FUNCTION_BLOCK "UTF8_TO_UNI"
{ S7_Optimized_Access := 'TRUE' }
VERSION : 0.1
   VAR_INPUT
      UTF8 : String[4];
   END_VAR

   VAR_OUTPUT
      UNICODE : Word;
   END_VAR

   VAR_TEMP
      TempDW : DWord;
      TempW : Array[0..3] of Word;
   END_VAR


BEGIN
	#TempDW := #UTF8[1];
	IF #TempDW < 16#80 THEN
	    #UNICODE := DWORD_TO_WORD(#TempDW AND 16#7F);
	ELSIF #TempDW >= 16#80 AND #TempDW < 16#C0 THEN
	    ;
	ELSIF #TempDW >= 16#C0 AND #TempDW < 16#E0 THEN
	    #TempDW := SHL(IN := #TempDW, N := 8);
	    #TempDW := #TempDW + BYTE_TO_WORD(#UTF8[2]);
	    #TempW[0] := DWORD_TO_WORD(SHR(IN:=#TempDW AND 16#1F00, N:=2));
	    #TempW[1] := DWORD_TO_WORD(#TempDW AND 16#3F);
	    #UNICODE := #TempW[0] + #TempW[1];
	ELSIF #TempDW >= 16#E0 AND #TempDW < 16#F0 THEN
	    #TempDW := SHL(IN := #TempDW, N := 8);
	    #TempDW := #TempDW + BYTE_TO_WORD(#UTF8[2]);
	    #TempDW := SHL(IN := #TempDW, N := 8);
	    #TempDW := #TempDW + BYTE_TO_WORD(#UTF8[3]);
	    #TempW[0] := DWORD_TO_WORD(SHR(IN:=#TempDW AND 16#0F0000, N:=4));
	    #TempW[1] := DWORD_TO_WORD(SHR(IN:=#TempDW AND 16#3F00, N:=2));
	    #TempW[2] := DWORD_TO_WORD(#TempDW AND 16#3F);
	    #UNICODE := #TempW[0] + #TempW[1] + #TempW[2];
	ELSIF #TempDW >= 16#F0 AND #TempDW < 16#F8 THEN
	    #TempDW := SHL(IN := #TempDW,  N := 8);
	    #TempDW := #TempDW + BYTE_TO_WORD(#UTF8[2]);
	    #TempDW := SHL(IN := #TempDW, N := 8);
	    #TempDW := #TempDW + BYTE_TO_WORD(#UTF8[3]);
	    #TempDW := SHL(IN := #TempDW,  N := 8);
	    #TempDW := #TempDW + BYTE_TO_WORD(#UTF8[4]);
	    #TempW[0] := DWORD_TO_WORD(SHR(IN:=#TempDW AND 16#7000000, N:=6));
	    #TempW[1] := DWORD_TO_WORD(SHR(IN:=#TempDW AND 16#3F0000, N:=4));
	    #TempW[2] := DWORD_TO_WORD(SHR(IN:=#TempDW AND 16#3F00, N:=2));
	    #TempW[3] := DWORD_TO_WORD(#TempDW AND 16#3F);
	    #UNICODE := #TempW[0] + #TempW[1] + #TempW[2] + #TempW[3];
	END_IF;
END_FUNCTION_BLOCK

FUNCTION_BLOCK "UNI_TO_GB2"
{ S7_Optimized_Access := 'TRUE' }
VERSION : 0.1
   VAR_INPUT
      UNICODE : Word;
   END_VAR

   VAR_OUTPUT
      GB2312 : Word;
   END_VAR

   VAR
      UNI : Array[0..7480] of Word := [16#00A4, 16#00A7, 16#00A8, 16#00B0, 16#00B1, 16#00B7, 16#00D7, 16#00E0, 16#00E1, 16#00E8, 16#00E9, 16#00EA, 16#00EC, 16#00ED, 16#00F2, 16#00F3, 16#00F7, 16#00F9, 16#00FA, 16#00FC, 16#0101, 16#0113, 16#011B, 16#012B, 16#0144, 16#0148, 16#014D, 16#016B, 16#01CE, 16#01D0, 16#01D2, 16#01D4, 16#01D6, 16#01D8, 16#01DA, 16#01DC, 16#0251, 16#0261, 16#02C7, 16#02C9, 16#0391, 16#0392, 16#0393, 16#0394, 16#0395, 16#0396, 16#0397, 16#0398, 16#0399, 16#039A, 16#039B, 16#039C, 16#039D, 16#039E, 16#039F, 16#03A0, 16#03A1, 16#03A3, 16#03A4, 16#03A5, 16#03A6, 16#03A7, 16#03A8, 16#03A9, 16#03B1, 16#03B2, 16#03B3, 16#03B4, 16#03B5, 16#03B6, 16#03B7, 16#03B8, 16#03B9, 16#03BA, 16#03BB, 16#03BC, 16#03BD, 16#03BE, 16#03BF, 16#03C0, 16#03C1, 16#03C3, 16#03C4, 16#03C5, 16#03C6, 16#03C7, 16#03C8, 16#03C9, 16#0401, 16#0410, 16#0411, 16#0412, 16#0413, 16#0414, 16#0415, 16#0416, 16#0417, 16#0418, 16#0419, 16#041A, 16#041B, 16#041C, 16#041D, 16#041E, 16#041F, 16#0420, 16#0421, 16#0422, 16#0423, 16#0424, 16#0425, 16#0426, 16#0427, 16#0428, 16#0429, 16#042A, 16#042B, 16#042C, 16#042D, 16#042E, 16#042F, 16#0430, 16#0431, 16#0432, 16#0433, 16#0434, 16#0435, 16#0436, 16#0437, 16#0438, 16#0439, 16#043A, 16#043B, 16#043C, 16#043D, 16#043E, 16#043F, 16#0440, 16#0441, 16#0442, 16#0443, 16#0444, 16#0445, 16#0446, 16#0447, 16#0448, 16#0449, 16#044A, 16#044B, 16#044C, 16#044D, 16#044E, 16#044F, 16#0451, 16#2014, 16#2016, 16#2018, 16#2019, 16#201C, 16#201D, 16#2026, 16#2030, 16#2032, 16#2033, 16#203B, 16#2103, 16#2116, 16#2160, 16#2161, 16#2162, 16#2163, 16#2164, 16#2165, 16#2166, 16#2167, 16#2168, 16#2169, 16#216A, 16#216B, 16#2170, 16#2171, 16#2172, 16#2173, 16#2174, 16#2175, 16#2176, 16#2177, 16#2178, 16#2179, 16#2190, 16#2191, 16#2192, 16#2193, 16#2208, 16#220F, 16#2211, 16#221A, 16#221D, 16#221E, 16#2220, 16#2225, 16#2227, 16#2228, 16#2229, 16#222A, 16#222B, 16#222E, 16#2234, 16#2235, 16#2236, 16#2237, 16#223D, 16#2248, 16#224C, 16#2260, 16#2261, 16#2264, 16#2265, 16#226E, 16#226F, 16#2299, 16#22A5, 16#2312, 16#2460, 16#2461, 16#2462, 16#2463, 16#2464, 16#2465, 16#2466, 16#2467, 16#2468, 16#2469, 16#2474, 16#2475, 16#2476, 16#2477, 16#2478, 16#2479, 16#247A, 16#247B, 16#247C, 16#247D, 16#247E, 16#247F, 16#2480, 16#2481, 16#2482, 16#2483, 16#2484, 16#2485, 16#2486, 16#2487, 16#2488, 16#2489, 16#248A, 16#248B, 16#248C, 16#248D, 16#248E, 16#248F, 16#2490, 16#2491, 16#2492, 16#2493, 16#2494, 16#2495, 16#2496, 16#2497, 16#2498, 16#2499, 16#249A, 16#249B, 16#2500, 16#2501, 16#2502, 16#2503, 16#2504, 16#2505, 16#2506, 16#2507, 16#2508, 16#2509, 16#250A, 16#250B, 16#250C, 16#250D, 16#250E, 16#250F, 16#2510, 16#2511, 16#2512, 16#2513, 16#2514, 16#2515, 16#2516, 16#2517, 16#2518, 16#2519, 16#251A, 16#251B, 16#251C, 16#251D, 16#251E, 16#251F, 16#2520, 16#2521, 16#2522, 16#2523, 16#2524, 16#2525, 16#2526, 16#2527, 16#2528, 16#2529, 16#252A, 16#252B, 16#252C, 16#252D, 16#252E, 16#252F, 16#2530, 16#2531, 16#2532, 16#2533, 16#2534, 16#2535, 16#2536, 16#2537, 16#2538, 16#2539, 16#253A, 16#253B, 16#253C, 16#253D, 16#253E, 16#253F, 16#2540, 16#2541, 16#2542, 16#2543, 16#2544, 16#2545, 16#2546, 16#2547, 16#2548, 16#2549, 16#254A, 16#254B, 16#25A0, 16#25A1, 16#25B2, 16#25B3, 16#25C6, 16#25C7, 16#25CB, 16#25CE, 16#25CF, 16#2605, 16#2606, 16#2640, 16#2642, 16#3000, 16#3001, 16#3002, 16#3003, 16#3005, 16#3008, 16#3009, 16#300A, 16#300B, 16#300C, 16#300D, 16#300E, 16#300F, 16#3010, 16#3011, 16#3013, 16#3014, 16#3015, 16#3016, 16#3017, 16#3041, 16#3042, 16#3043, 16#3044, 16#3045, 16#3046, 16#3047, 16#3048, 16#3049, 16#304A, 16#304B, 16#304C, 16#304D, 16#304E, 16#304F, 16#3050, 16#3051, 16#3052, 16#3053, 16#3054, 16#3055, 16#3056, 16#3057, 16#3058, 16#3059, 16#305A, 16#305B, 16#305C, 16#305D, 16#305E, 16#305F, 16#3060, 16#3061, 16#3062, 16#3063, 16#3064, 16#3065, 16#3066, 16#3067, 16#3068, 16#3069, 16#306A, 16#306B, 16#306C, 16#306D, 16#306E, 16#306F, 16#3070, 16#3071, 16#3072, 16#3073, 16#3074, 16#3075, 16#3076, 16#3077, 16#3078, 16#3079, 16#307A, 16#307B, 16#307C, 16#307D, 16#307E, 16#307F, 16#3080, 16#3081, 16#3082, 16#3083, 16#3084, 16#3085, 16#3086, 16#3087, 16#3088, 16#3089, 16#308A, 16#308B, 16#308C, 16#308D, 16#308E, 16#308F, 16#3090, 16#3091, 16#3092, 16#3093, 16#30A1, 16#30A2, 16#30A3, 16#30A4, 16#30A5, 16#30A6, 16#30A7, 16#30A8, 16#30A9, 16#30AA, 16#30AB, 16#30AC, 16#30AD, 16#30AE, 16#30AF, 16#30B0, 16#30B1, 16#30B2, 16#30B3, 16#30B4, 16#30B5, 16#30B6, 16#30B7, 16#30B8, 16#30B9, 16#30BA, 16#30BB, 16#30BC, 16#30BD, 16#30BE, 16#30BF, 16#30C0, 16#30C1, 16#30C2, 16#30C3, 16#30C4, 16#30C5, 16#30C6, 16#30C7, 16#30C8, 16#30C9, 16#30CA, 16#30CB, 16#30CC, 16#30CD, 16#30CE, 16#30CF, 16#30D0, 16#30D1, 16#30D2, 16#30D3, 16#30D4, 16#30D5, 16#30D6, 16#30D7, 16#30D8, 16#30D9, 16#30DA, 16#30DB, 16#30DC, 16#30DD, 16#30DE, 16#30DF, 16#30E0, 16#30E1, 16#30E2, 16#30E3, 16#30E4, 16#30E5, 16#30E6, 16#30E7, 16#30E8, 16#30E9, 16#30EA, 16#30EB, 16#30EC, 16#30ED, 16#30EE, 16#30EF, 16#30F0, 16#30F1, 16#30F2, 16#30F3, 16#30F4, 16#30F5, 16#30F6, 16#3105, 16#3106, 16#3107, 16#3108, 16#3109, 16#310A, 16#310B, 16#310C, 16#310D, 16#310E, 16#310F, 16#3110, 16#3111, 16#3112, 16#3113, 16#3114, 16#3115, 16#3116, 16#3117, 16#3118, 16#3119, 16#311A, 16#311B, 16#311C, 16#311D, 16#311E, 16#311F, 16#3120, 16#3121, 16#3122, 16#3123, 16#3124, 16#3125, 16#3126, 16#3127, 16#3128, 16#3129, 16#3220, 16#3221, 16#3222, 16#3223, 16#3224, 16#3225, 16#3226, 16#3227, 16#3228, 16#3229, 16#4E00, 16#4E01, 16#4E03, 16#4E07, 16#4E08, 16#4E09, 16#4E0A, 16#4E0B, 16#4E0C, 16#4E0D, 16#4E0E, 16#4E10, 16#4E11, 16#4E13, 16#4E14, 16#4E15, 16#4E16, 16#4E18, 16#4E19, 16#4E1A, 16#4E1B, 16#4E1C, 16#4E1D, 16#4E1E, 16#4E22, 16#4E24, 16#4E25, 16#4E27, 16#4E28, 16#4E2A, 16#4E2B, 16#4E2C, 16#4E2D, 16#4E30, 16#4E32, 16#4E34, 16#4E36, 16#4E38, 16#4E39, 16#4E3A, 16#4E3B, 16#4E3D, 16#4E3E, 16#4E3F, 16#4E43, 16#4E45, 16#4E47, 16#4E48, 16#4E49, 16#4E4B, 16#4E4C, 16#4E4D, 16#4E4E, 16#4E4F, 16#4E50, 16#4E52, 16#4E53, 16#4E54, 16#4E56, 16#4E58, 16#4E59, 16#4E5C, 16#4E5D, 16#4E5E, 16#4E5F, 16#4E60, 16#4E61, 16#4E66, 16#4E69, 16#4E70, 16#4E71, 16#4E73, 16#4E7E, 16#4E86, 16#4E88, 16#4E89, 16#4E8B, 16#4E8C, 16#4E8D, 16#4E8E, 16#4E8F, 16#4E91, 16#4E92, 16#4E93, 16#4E94, 16#4E95, 16#4E98, 16#4E9A, 16#4E9B, 16#4E9F, 16#4EA0, 16#4EA1, 16#4EA2, 16#4EA4, 16#4EA5, 16#4EA6, 16#4EA7, 16#4EA8, 16#4EA9, 16#4EAB, 16#4EAC, 16#4EAD, 16#4EAE, 16#4EB2, 16#4EB3, 16#4EB5, 16#4EBA, 16#4EBB, 16#4EBF, 16#4EC0, 16#4EC1, 16#4EC2, 16#4EC3, 16#4EC4, 16#4EC5, 16#4EC6, 16#4EC7, 16#4EC9, 16#4ECA, 16#4ECB, 16#4ECD, 16#4ECE, 16#4ED1, 16#4ED3, 16#4ED4, 16#4ED5, 16#4ED6, 16#4ED7, 16#4ED8, 16#4ED9, 16#4EDD, 16#4EDE, 16#4EDF, 16#4EE1, 16#4EE3, 16#4EE4, 16#4EE5, 16#4EE8, 16#4EEA, 16#4EEB, 16#4EEC, 16#4EF0, 16#4EF2, 16#4EF3, 16#4EF5, 16#4EF6, 16#4EF7, 16#4EFB, 16#4EFD, 16#4EFF, 16#4F01, 16#4F09, 16#4F0A, 16#4F0D, 16#4F0E, 16#4F0F, 16#4F10, 16#4F11, 16#4F17, 16#4F18, 16#4F19, 16#4F1A, 16#4F1B, 16#4F1E, 16#4F1F, 16#4F20, 16#4F22, 16#4F24, 16#4F25, 16#4F26, 16#4F27, 16#4F2A, 16#4F2B, 16#4F2F, 16#4F30, 16#4F32, 16#4F34, 16#4F36, 16#4F38, 16#4F3A, 16#4F3C, 16#4F3D, 16#4F43, 16#4F46, 16#4F4D, 16#4F4E, 16#4F4F, 16#4F50, 16#4F51, 16#4F53, 16#4F55, 16#4F57, 16#4F58, 16#4F59, 16#4F5A, 16#4F5B, 16#4F5C, 16#4F5D, 16#4F5E, 16#4F5F, 16#4F60, 16#4F63, 16#4F64, 16#4F65, 16#4F67, 16#4F69, 16#4F6C, 16#4F6F, 16#4F70, 16#4F73, 16#4F74, 16#4F76, 16#4F7B, 16#4F7C, 16#4F7E, 16#4F7F, 16#4F83, 16#4F84, 16#4F88, 16#4F89, 16#4F8B, 16#4F8D, 16#4F8F, 16#4F91, 16#4F94, 16#4F97, 16#4F9B, 16#4F9D, 16#4FA0, 16#4FA3, 16#4FA5, 16#4FA6, 16#4FA7, 16#4FA8, 16#4FA9, 16#4FAA, 16#4FAC, 16#4FAE, 16#4FAF, 16#4FB5, 16#4FBF, 16#4FC3, 16#4FC4, 16#4FC5, 16#4FCA, 16#4FCE, 16#4FCF, 16#4FD0, 16#4FD1, 16#4FD7, 16#4FD8, 16#4FDA, 16#4FDC, 16#4FDD, 16#4FDE, 16#4FDF, 16#4FE1, 16#4FE3, 16#4FE6, 16#4FE8, 16#4FE9, 16#4FEA, 16#4FED, 16#4FEE, 16#4FEF, 16#4FF1, 16#4FF3, 16#4FF8, 16#4FFA, 16#4FFE, 16#500C, 16#500D, 16#500F, 16#5012, 16#5014, 16#5018, 16#5019, 16#501A, 16#501C, 16#501F, 16#5021, 16#5025, 16#5026, 16#5028, 16#5029, 16#502A, 16#502C, 16#502D, 16#502E, 16#503A, 16#503C, 16#503E, 16#5043, 16#5047, 16#5048, 16#504C, 16#504E, 16#504F, 16#5055, 16#505A, 16#505C, 16#5065, 16#506C, 16#5076, 16#5077, 16#507B, 16#507E, 16#507F, 16#5080, 16#5085, 16#5088, 16#508D, 16#50A3, 16#50A5, 16#50A7, 16#50A8, 16#50A9, 16#50AC, 16#50B2, 16#50BA, 16#50BB, 16#50CF, 16#50D6, 16#50DA, 16#50E6, 16#50E7, 16#50EC, 16#50ED, 16#50EE, 16#50F3, 16#50F5, 16#50FB, 16#5106, 16#5107, 16#510B, 16#5112, 16#5121, 16#513F, 16#5140, 16#5141, 16#5143, 16#5144, 16#5145, 16#5146, 16#5148, 16#5149, 16#514B, 16#514D, 16#5151, 16#5154, 16#5155, 16#5156, 16#515A, 16#515C, 16#5162, 16#5165, 16#5168, 16#516B, 16#516C, 16#516D, 16#516E, 16#5170, 16#5171, 16#5173, 16#5174, 16#5175, 16#5176, 16#5177, 16#5178, 16#5179, 16#517B, 16#517C, 16#517D, 16#5180, 16#5181, 16#5182, 16#5185, 16#5188, 16#5189, 16#518C, 16#518D, 16#5192, 16#5195, 16#5196, 16#5197, 16#5199, 16#519B, 16#519C, 16#51A0, 16#51A2, 16#51A4, 16#51A5, 16#51AB, 16#51AC, 16#51AF, 16#51B0, 16#51B1, 16#51B2, 16#51B3, 16#51B5, 16#51B6, 16#51B7, 16#51BB, 16#51BC, 16#51BD, 16#51C0, 16#51C4, 16#51C6, 16#51C7, 16#51C9, 16#51CB, 16#51CC, 16#51CF, 16#51D1, 16#51DB, 16#51DD, 16#51E0, 16#51E1, 16#51E4, 16#51EB, 16#51ED, 16#51EF, 16#51F0, 16#51F3, 16#51F5, 16#51F6, 16#51F8, 16#51F9, 16#51FA, 16#51FB, 16#51FC, 16#51FD, 16#51FF, 16#5200, 16#5201, 16#5202, 16#5203, 16#5206, 16#5207, 16#5208, 16#520A, 16#520D, 16#520E, 16#5211, 16#5212, 16#5216, 16#5217, 16#5218, 16#5219, 16#521A, 16#521B, 16#521D, 16#5220, 16#5224, 16#5228, 16#5229, 16#522B, 16#522D, 16#522E, 16#5230, 16#5233, 16#5236, 16#5237, 16#5238, 16#5239, 16#523A, 16#523B, 16#523D, 16#523F, 16#5240, 16#5241, 16#5242, 16#5243, 16#524A, 16#524C, 16#524D, 16#5250, 16#5251, 16#5254, 16#5256, 16#525C, 16#525E, 16#5261, 16#5265, 16#5267, 16#5269, 16#526A, 16#526F, 16#5272, 16#527D, 16#527F, 16#5281, 16#5282, 16#5288, 16#5290, 16#5293, 16#529B, 16#529D, 16#529E, 16#529F, 16#52A0, 16#52A1, 16#52A2, 16#52A3, 16#52A8, 16#52A9, 16#52AA, 16#52AB, 16#52AC, 16#52AD, 16#52B1, 16#52B2, 16#52B3, 16#52BE, 16#52BF, 16#52C3, 16#52C7, 16#52C9, 16#52CB, 16#52D0, 16#52D2, 16#52D6, 16#52D8, 16#52DF, 16#52E4, 16#52F0, 16#52F9, 16#52FA, 16#52FE, 16#52FF, 16#5300, 16#5305, 16#5306, 16#5308, 16#530D, 16#530F, 16#5310, 16#5315, 16#5316, 16#5317, 16#5319, 16#531A, 16#531D, 16#5320, 16#5321, 16#5323, 16#5326, 16#532A, 16#532E, 16#5339, 16#533A, 16#533B, 16#533E, 16#533F, 16#5341, 16#5343, 16#5345, 16#5347, 16#5348, 16#5349, 16#534A, 16#534E, 16#534F, 16#5351, 16#5352, 16#5353, 16#5355, 16#5356, 16#5357, 16#535A, 16#535C, 16#535E, 16#535F, 16#5360, 16#5361, 16#5362, 16#5363, 16#5364, 16#5366, 16#5367, 16#5369, 16#536B, 16#536E, 16#536F, 16#5370, 16#5371, 16#5373, 16#5374, 16#5375, 16#5377, 16#5378, 16#537A, 16#537F, 16#5382, 16#5384, 16#5385, 16#5386, 16#5389, 16#538B, 16#538C, 16#538D, 16#5395, 16#5398, 16#539A, 16#539D, 16#539F, 16#53A2, 16#53A3, 16#53A5, 16#53A6, 16#53A8, 16#53A9, 16#53AE, 16#53B6, 16#53BB, 16#53BF, 16#53C1, 16#53C2, 16#53C8, 16#53C9, 16#53CA, 16#53CB, 16#53CC, 16#53CD, 16#53D1, 16#53D4, 16#53D6, 16#53D7, 16#53D8, 16#53D9, 16#53DB, 16#53DF, 16#53E0, 16#53E3, 16#53E4, 16#53E5, 16#53E6, 16#53E8, 16#53E9, 16#53EA, 16#53EB, 16#53EC, 16#53ED, 16#53EE, 16#53EF, 16#53F0, 16#53F1, 16#53F2, 16#53F3, 16#53F5, 16#53F6, 16#53F7, 16#53F8, 16#53F9, 16#53FB, 16#53FC, 16#53FD, 16#5401, 16#5403, 16#5404, 16#5406, 16#5408, 16#5409, 16#540A, 16#540C, 16#540D, 16#540E, 16#540F, 16#5410, 16#5411, 16#5412, 16#5413, 16#5415, 16#5416, 16#5417, 16#541B, 16#541D, 16#541E, 16#541F, 16#5420, 16#5421, 16#5423, 16#5426, 16#5427, 16#5428, 16#5429, 16#542B, 16#542C, 16#542D, 16#542E, 16#542F, 16#5431, 16#5432, 16#5434, 16#5435, 16#5438, 16#5439, 16#543B, 16#543C, 16#543E, 16#5440, 16#5443, 16#5446, 16#5448, 16#544A, 16#544B, 16#5450, 16#5452, 16#5453, 16#5454, 16#5455, 16#5456, 16#5457, 16#5458, 16#5459, 16#545B, 16#545C, 16#5462, 16#5464, 16#5466, 16#5468, 16#5471, 16#5472, 16#5473, 16#5475, 16#5476, 16#5477, 16#5478, 16#547B, 16#547C, 16#547D, 16#5480, 16#5482, 16#5484, 16#5486, 16#548B, 16#548C, 16#548E, 16#548F, 16#5490, 16#5492, 16#5494, 16#5495, 16#5496, 16#5499, 16#549A, 16#549B, 16#549D, 16#54A3, 16#54A4, 16#54A6, 16#54A7, 16#54A8, 16#54A9, 16#54AA, 16#54AB, 16#54AC, 16#54AD, 16#54AF, 16#54B1, 16#54B3, 16#54B4, 16#54B8, 16#54BB, 16#54BD, 16#54BF, 16#54C0, 16#54C1, 16#54C2, 16#54C4, 16#54C6, 16#54C7, 16#54C8, 16#54C9, 16#54CC, 16#54CD, 16#54CE, 16#54CF, 16#54D0, 16#54D1, 16#54D2, 16#54D3, 16#54D4, 16#54D5, 16#54D7, 16#54D9, 16#54DA, 16#54DC, 16#54DD, 16#54DE, 16#54DF, 16#54E5, 16#54E6, 16#54E7, 16#54E8, 16#54E9, 16#54EA, 16#54ED, 16#54EE, 16#54F2, 16#54F3, 16#54FA, 16#54FC, 16#54FD, 16#54FF, 16#5501, 16#5506, 16#5507, 16#5509, 16#550F, 16#5510, 16#5511, 16#5514, 16#551B, 16#5520, 16#5522, 16#5523, 16#5524, 16#5527, 16#552A, 16#552C, 16#552E, 16#552F, 16#5530, 16#5531, 16#5533, 16#5537, 16#553C, 16#553E, 16#553F, 16#5541, 16#5543, 16#5544, 16#5546, 16#5549, 16#554A, 16#5550, 16#5555, 16#5556, 16#555C, 16#5561, 16#5564, 16#5565, 16#5566, 16#5567, 16#556A, 16#556C, 16#556D, 16#556E, 16#5575, 16#5576, 16#5577, 16#5578, 16#557B, 16#557C, 16#557E, 16#5580, 16#5581, 16#5582, 16#5583, 16#5584, 16#5587, 16#5588, 16#5589, 16#558A, 16#558B, 16#558F, 16#5591, 16#5594, 16#5598, 16#5599, 16#559C, 16#559D, 16#559F, 16#55A7, 16#55B1, 16#55B3, 16#55B5, 16#55B7, 16#55B9, 16#55BB, 16#55BD, 16#55BE, 16#55C4, 16#55C5, 16#55C9, 16#55CC, 16#55CD, 16#55D1, 16#55D2, 16#55D3, 16#55D4, 16#55D6, 16#55DC, 16#55DD, 16#55DF, 16#55E1, 16#55E3, 16#55E4, 16#55E5, 16#55E6, 16#55E8, 16#55EA, 16#55EB, 16#55EC, 16#55EF, 16#55F2, 16#55F3, 16#55F5, 16#55F7, 16#55FD, 16#55FE, 16#5600, 16#5601, 16#5608, 16#5609, 16#560C, 16#560E, 16#560F, 16#5618, 16#561B, 16#561E, 16#561F, 16#5623, 16#5624, 16#5627, 16#562C, 16#562D, 16#5631, 16#5632, 16#5634, 16#5636, 16#5639, 16#563B, 16#563F, 16#564C, 16#564D, 16#564E, 16#5654, 16#5657, 16#5658, 16#5659, 16#565C, 16#5662, 16#5664, 16#5668, 16#5669, 16#566A, 16#566B, 16#566C, 16#5671, 16#5676, 16#567B, 16#567C, 16#5685, 16#5686, 16#568E, 16#568F, 16#5693, 16#56A3, 16#56AF, 16#56B7, 16#56BC, 16#56CA, 16#56D4, 16#56D7, 16#56DA, 16#56DB, 16#56DD, 16#56DE, 16#56DF, 16#56E0, 16#56E1, 16#56E2, 16#56E4, 16#56EB, 16#56ED, 16#56F0, 16#56F1, 16#56F4, 16#56F5, 16#56F9, 16#56FA, 16#56FD, 16#56FE, 16#56FF, 16#5703, 16#5704, 16#5706, 16#5708, 16#5709, 16#570A, 16#571C, 16#571F, 16#5723, 16#5728, 16#5729, 16#572A, 16#572C, 16#572D, 16#572E, 16#572F, 16#5730, 16#5733, 16#5739, 16#573A, 16#573B, 16#573E, 16#5740, 16#5742, 16#5747, 16#574A, 16#574C, 16#574D, 16#574E, 16#574F, 16#5750, 16#5751, 16#5757, 16#575A, 16#575B, 16#575C, 16#575D, 16#575E, 16#575F, 16#5760, 16#5761, 16#5764, 16#5766, 16#5768, 16#5769, 16#576A, 16#576B, 16#576D, 16#576F, 16#5773, 16#5776, 16#5777, 16#577B, 16#577C, 16#5782, 16#5783, 16#5784, 16#5785, 16#5786, 16#578B, 16#578C, 16#5792, 16#5793, 16#579B, 16#57A0, 16#57A1, 16#57A2, 16#57A3, 16#57A4, 16#57A6, 16#57A7, 16#57A9, 16#57AB, 16#57AD, 16#57AE, 16#57B2, 16#57B4, 16#57B8, 16#57C2, 16#57C3, 16#57CB, 16#57CE, 16#57CF, 16#57D2, 16#57D4, 16#57D5, 16#57D8, 16#57D9, 16#57DA, 16#57DD, 16#57DF, 16#57E0, 16#57E4, 16#57ED, 16#57EF, 16#57F4, 16#57F8, 16#57F9, 16#57FA, 16#57FD, 16#5800, 16#5802, 16#5806, 16#5807, 16#580B, 16#580D, 16#5811, 16#5815, 16#5819, 16#581E, 16#5820, 16#5821, 16#5824, 16#582A, 16#5830, 16#5835, 16#5844, 16#584C, 16#584D, 16#5851, 16#5854, 16#5858, 16#585E, 16#5865, 16#586B, 16#586C, 16#587E, 16#5880, 16#5881, 16#5883, 16#5885, 16#5889, 16#5892, 16#5893, 16#5899, 16#589A, 16#589E, 16#589F, 16#58A8, 16#58A9, 16#58BC, 16#58C1, 16#58C5, 16#58D1, 16#58D5, 16#58E4, 16#58EB, 16#58EC, 16#58EE, 16#58F0, 16#58F3, 16#58F6, 16#58F9, 16#5902, 16#5904, 16#5907, 16#590D, 16#590F, 16#5914, 16#5915, 16#5916, 16#5919, 16#591A, 16#591C, 16#591F, 16#5924, 16#5925, 16#5927, 16#5929, 16#592A, 16#592B, 16#592D, 16#592E, 16#592F, 16#5931, 16#5934, 16#5937, 16#5938, 16#5939, 16#593A, 16#593C, 16#5941, 16#5942, 16#5944, 16#5947, 16#5948, 16#5949, 16#594B, 16#594E, 16#594F, 16#5951, 16#5954, 16#5955, 16#5956, 16#5957, 16#5958, 16#595A, 16#5960, 16#5962, 16#5965, 16#5973, 16#5974, 16#5976, 16#5978, 16#5979, 16#597D, 16#5981, 16#5982, 16#5983, 16#5984, 16#5986, 16#5987, 16#5988, 16#598A, 16#598D, 16#5992, 16#5993, 16#5996, 16#5997, 16#5999, 16#599E, 16#59A3, 16#59A4, 16#59A5, 16#59A8, 16#59A9, 16#59AA, 16#59AB, 16#59AE, 16#59AF, 16#59B2, 16#59B9, 16#59BB, 16#59BE, 16#59C6, 16#59CA, 16#59CB, 16#59D0, 16#59D1, 16#59D2, 16#59D3, 16#59D4, 16#59D7, 16#59D8, 16#59DA, 16#59DC, 16#59DD, 16#59E3, 16#59E5, 16#59E8, 16#59EC, 16#59F9, 16#59FB, 16#59FF, 16#5A01, 16#5A03, 16#5A04, 16#5A05, 16#5A06, 16#5A07, 16#5A08, 16#5A09, 16#5A0C, 16#5A11, 16#5A13, 16#5A18, 16#5A1C, 16#5A1F, 16#5A20, 16#5A23, 16#5A25, 16#5A29, 16#5A31, 16#5A32, 16#5A34, 16#5A36, 16#5A3C, 16#5A40, 16#5A46, 16#5A49, 16#5A4A, 16#5A55, 16#5A5A, 16#5A62, 16#5A67, 16#5A6A, 16#5A74, 16#5A75, 16#5A76, 16#5A77, 16#5A7A, 16#5A7F, 16#5A92, 16#5A9A, 16#5A9B, 16#5AAA, 16#5AB2, 16#5AB3, 16#5AB5, 16#5AB8, 16#5ABE, 16#5AC1, 16#5AC2, 16#5AC9, 16#5ACC, 16#5AD2, 16#5AD4, 16#5AD6, 16#5AD8, 16#5ADC, 16#5AE0, 16#5AE1, 16#5AE3, 16#5AE6, 16#5AE9, 16#5AEB, 16#5AF1, 16#5B09, 16#5B16, 16#5B17, 16#5B32, 16#5B34, 16#5B37, 16#5B40, 16#5B50, 16#5B51, 16#5B53, 16#5B54, 16#5B55, 16#5B57, 16#5B58, 16#5B59, 16#5B5A, 16#5B5B, 16#5B5C, 16#5B5D, 16#5B5F, 16#5B62, 16#5B63, 16#5B64, 16#5B65, 16#5B66, 16#5B69, 16#5B6A, 16#5B6C, 16#5B70, 16#5B71, 16#5B73, 16#5B75, 16#5B7A, 16#5B7D, 16#5B80, 16#5B81, 16#5B83, 16#5B84, 16#5B85, 16#5B87, 16#5B88, 16#5B89, 16#5B8B, 16#5B8C, 16#5B8F, 16#5B93, 16#5B95, 16#5B97, 16#5B98, 16#5B99, 16#5B9A, 16#5B9B, 16#5B9C, 16#5B9D, 16#5B9E, 16#5BA0, 16#5BA1, 16#5BA2, 16#5BA3, 16#5BA4, 16#5BA5, 16#5BA6, 16#5BAA, 16#5BAB, 16#5BB0, 16#5BB3, 16#5BB4, 16#5BB5, 16#5BB6, 16#5BB8, 16#5BB9, 16#5BBD, 16#5BBE, 16#5BBF, 16#5BC2, 16#5BC4, 16#5BC5, 16#5BC6, 16#5BC7, 16#5BCC, 16#5BD0, 16#5BD2, 16#5BD3, 16#5BDD, 16#5BDE, 16#5BDF, 16#5BE1, 16#5BE4, 16#5BE5, 16#5BE8, 16#5BEE, 16#5BF0, 16#5BF8, 16#5BF9, 16#5BFA, 16#5BFB, 16#5BFC, 16#5BFF, 16#5C01, 16#5C04, 16#5C06, 16#5C09, 16#5C0A, 16#5C0F, 16#5C11, 16#5C14, 16#5C15, 16#5C16, 16#5C18, 16#5C1A, 16#5C1C, 16#5C1D, 16#5C22, 16#5C24, 16#5C25, 16#5C27, 16#5C2C, 16#5C31, 16#5C34, 16#5C38, 16#5C39, 16#5C3A, 16#5C3B, 16#5C3C, 16#5C3D, 16#5C3E, 16#5C3F, 16#5C40, 16#5C41, 16#5C42, 16#5C45, 16#5C48, 16#5C49, 16#5C4A, 16#5C4B, 16#5C4E, 16#5C4F, 16#5C50, 16#5C51, 16#5C55, 16#5C59, 16#5C5E, 16#5C60, 16#5C61, 16#5C63, 16#5C65, 16#5C66, 16#5C6E, 16#5C6F, 16#5C71, 16#5C79, 16#5C7A, 16#5C7F, 16#5C81, 16#5C82, 16#5C88, 16#5C8C, 16#5C8D, 16#5C90, 16#5C91, 16#5C94, 16#5C96, 16#5C97, 16#5C98, 16#5C99, 16#5C9A, 16#5C9B, 16#5C9C, 16#5CA2, 16#5CA3, 16#5CA9, 16#5CAB, 16#5CAC, 16#5CAD, 16#5CB1, 16#5CB3, 16#5CB5, 16#5CB7, 16#5CB8, 16#5CBD, 16#5CBF, 16#5CC1, 16#5CC4, 16#5CCB, 16#5CD2, 16#5CD9, 16#5CE1, 16#5CE4, 16#5CE5, 16#5CE6, 16#5CE8, 16#5CEA, 16#5CED, 16#5CF0, 16#5CFB, 16#5D02, 16#5D03, 16#5D06, 16#5D07, 16#5D0E, 16#5D14, 16#5D16, 16#5D1B, 16#5D1E, 16#5D24, 16#5D26, 16#5D27, 16#5D29, 16#5D2D, 16#5D2E, 16#5D34, 16#5D3D, 16#5D3E, 16#5D47, 16#5D4A, 16#5D4B, 16#5D4C, 16#5D58, 16#5D5B, 16#5D5D, 16#5D69, 16#5D6B, 16#5D6C, 16#5D6F, 16#5D74, 16#5D82, 16#5D99, 16#5D9D, 16#5DB7, 16#5DC5, 16#5DCD, 16#5DDB, 16#5DDD, 16#5DDE, 16#5DE1, 16#5DE2, 16#5DE5, 16#5DE6, 16#5DE7, 16#5DE8, 16#5DE9, 16#5DEB, 16#5DEE, 16#5DEF, 16#5DF1, 16#5DF2, 16#5DF3, 16#5DF4, 16#5DF7, 16#5DFD, 16#5DFE, 16#5E01, 16#5E02, 16#5E03, 16#5E05, 16#5E06, 16#5E08, 16#5E0C, 16#5E0F, 16#5E10, 16#5E11, 16#5E14, 16#5E15, 16#5E16, 16#5E18, 16#5E19, 16#5E1A, 16#5E1B, 16#5E1C, 16#5E1D, 16#5E26, 16#5E27, 16#5E2D, 16#5E2E, 16#5E31, 16#5E37, 16#5E38, 16#5E3B, 16#5E3C, 16#5E3D, 16#5E42, 16#5E44, 16#5E45, 16#5E4C, 16#5E54, 16#5E55, 16#5E5B, 16#5E5E, 16#5E61, 16#5E62, 16#5E72, 16#5E73, 16#5E74, 16#5E76, 16#5E78, 16#5E7A, 16#5E7B, 16#5E7C, 16#5E7D, 16#5E7F, 16#5E80, 16#5E84, 16#5E86, 16#5E87, 16#5E8A, 16#5E8B, 16#5E8F, 16#5E90, 16#5E91, 16#5E93, 16#5E94, 16#5E95, 16#5E96, 16#5E97, 16#5E99, 16#5E9A, 16#5E9C, 16#5E9E, 16#5E9F, 16#5EA0, 16#5EA5, 16#5EA6, 16#5EA7, 16#5EAD, 16#5EB3, 16#5EB5, 16#5EB6, 16#5EB7, 16#5EB8, 16#5EB9, 16#5EBE, 16#5EC9, 16#5ECA, 16#5ED1, 16#5ED2, 16#5ED3, 16#5ED6, 16#5EDB, 16#5EE8, 16#5EEA, 16#5EF4, 16#5EF6, 16#5EF7, 16#5EFA, 16#5EFE, 16#5EFF, 16#5F00, 16#5F01, 16#5F02, 16#5F03, 16#5F04, 16#5F08, 16#5F0A, 16#5F0B, 16#5F0F, 16#5F11, 16#5F13, 16#5F15, 16#5F17, 16#5F18, 16#5F1B, 16#5F1F, 16#5F20, 16#5F25, 16#5F26, 16#5F27, 16#5F29, 16#5F2A, 16#5F2D, 16#5F2F, 16#5F31, 16#5F39, 16#5F3A, 16#5F3C, 16#5F40, 16#5F50, 16#5F52, 16#5F53, 16#5F55, 16#5F56, 16#5F57, 16#5F58, 16#5F5D, 16#5F61, 16#5F62, 16#5F64, 16#5F66, 16#5F69, 16#5F6A, 16#5F6C, 16#5F6D, 16#5F70, 16#5F71, 16#5F73, 16#5F77, 16#5F79, 16#5F7B, 16#5F7C, 16#5F80, 16#5F81, 16#5F82, 16#5F84, 16#5F85, 16#5F87, 16#5F88, 16#5F89, 16#5F8A, 16#5F8B, 16#5F8C, 16#5F90, 16#5F92, 16#5F95, 16#5F97, 16#5F98, 16#5F99, 16#5F9C, 16#5FA1, 16#5FA8, 16#5FAA, 16#5FAD, 16#5FAE, 16#5FB5, 16#5FB7, 16#5FBC, 16#5FBD, 16#5FC3, 16#5FC4, 16#5FC5, 16#5FC6, 16#5FC9, 16#5FCC, 16#5FCD, 16#5FCF, 16#5FD0, 16#5FD1, 16#5FD2, 16#5FD6, 16#5FD7, 16#5FD8, 16#5FD9, 16#5FDD, 16#5FE0, 16#5FE1, 16#5FE4, 16#5FE7, 16#5FEA, 16#5FEB, 16#5FED, 16#5FEE, 16#5FF1, 16#5FF5, 16#5FF8, 16#5FFB, 16#5FFD, 16#5FFE, 16#5FFF, 16#6000, 16#6001, 16#6002, 16#6003, 16#6004, 16#6005, 16#6006, 16#600A, 16#600D, 16#600E, 16#600F, 16#6012, 16#6014, 16#6015, 16#6016, 16#6019, 16#601B, 16#601C, 16#601D, 16#6020, 16#6021, 16#6025, 16#6026, 16#6027, 16#6028, 16#6029, 16#602A, 16#602B, 16#602F, 16#6035, 16#603B, 16#603C, 16#603F, 16#6041, 16#6042, 16#6043, 16#604B, 16#604D, 16#6050, 16#6052, 16#6055, 16#6059, 16#605A, 16#605D, 16#6062, 16#6063, 16#6064, 16#6067, 16#6068, 16#6069, 16#606A, 16#606B, 16#606C, 16#606D, 16#606F, 16#6070, 16#6073, 16#6076, 16#6078, 16#6079, 16#607A, 16#607B, 16#607C, 16#607D, 16#607F, 16#6083, 16#6084, 16#6089, 16#608C, 16#608D, 16#6092, 16#6094, 16#6096, 16#609A, 16#609B, 16#609D, 16#609F, 16#60A0, 16#60A3, 16#60A6, 16#60A8, 16#60AB, 16#60AC, 16#60AD, 16#60AF, 16#60B1, 16#60B2, 16#60B4, 16#60B8, 16#60BB, 16#60BC, 16#60C5, 16#60C6, 16#60CA, 16#60CB, 16#60D1, 16#60D5, 16#60D8, 16#60DA, 16#60DC, 16#60DD, 16#60DF, 16#60E0, 16#60E6, 16#60E7, 16#60E8, 16#60E9, 16#60EB, 16#60EC, 16#60ED, 16#60EE, 16#60EF, 16#60F0, 16#60F3, 16#60F4, 16#60F6, 16#60F9, 16#60FA, 16#6100, 16#6101, 16#6106, 16#6108, 16#6109, 16#610D, 16#610E, 16#610F, 16#6115, 16#611A, 16#611F, 16#6120, 16#6123, 16#6124, 16#6126, 16#6127, 16#612B, 16#613F, 16#6148, 16#614A, 16#614C, 16#614E, 16#6151, 16#6155, 16#615D, 16#6162, 16#6167, 16#6168, 16#6170, 16#6175, 16#6177, 16#618B, 16#618E, 16#6194, 16#619D, 16#61A7, 16#61A8, 16#61A9, 16#61AC, 16#61B7, 16#61BE, 16#61C2, 16#61C8, 16#61CA, 16#61CB, 16#61D1, 16#61D2, 16#61D4, 16#61E6, 16#61F5, 16#61FF, 16#6206, 16#6208, 16#620A, 16#620B, 16#620C, 16#620D, 16#620E, 16#620F, 16#6210, 16#6211, 16#6212, 16#6215, 16#6216, 16#6217, 16#6218, 16#621A, 16#621B, 16#621F, 16#6221, 16#6222, 16#6224, 16#6225, 16#622A, 16#622C, 16#622E, 16#6233, 16#6234, 16#6237, 16#623D, 16#623E, 16#623F, 16#6240, 16#6241, 16#6243, 16#6247, 16#6248, 16#6249, 16#624B, 16#624C, 16#624D, 16#624E, 16#6251, 16#6252, 16#6253, 16#6254, 16#6258, 16#625B, 16#6263, 16#6266, 16#6267, 16#6269, 16#626A, 16#626B, 16#626C, 16#626D, 16#626E, 16#626F, 16#6270, 16#6273, 16#6276, 16#6279, 16#627C, 16#627E, 16#627F, 16#6280, 16#6284, 16#6289, 16#628A, 16#6291, 16#6292, 16#6293, 16#6295, 16#6296, 16#6297, 16#6298, 16#629A, 16#629B, 16#629F, 16#62A0, 16#62A1, 16#62A2, 16#62A4, 16#62A5, 16#62A8, 16#62AB, 16#62AC, 16#62B1, 16#62B5, 16#62B9, 16#62BB, 16#62BC, 16#62BD, 16#62BF, 16#62C2, 16#62C4, 16#62C5, 16#62C6, 16#62C7, 16#62C8, 16#62C9, 16#62CA, 16#62CC, 16#62CD, 16#62CE, 16#62D0, 16#62D2, 16#62D3, 16#62D4, 16#62D6, 16#62D7, 16#62D8, 16#62D9, 16#62DA, 16#62DB, 16#62DC, 16#62DF, 16#62E2, 16#62E3, 16#62E5, 16#62E6, 16#62E7, 16#62E8, 16#62E9, 16#62EC, 16#62ED, 16#62EE, 16#62EF, 16#62F1, 16#62F3, 16#62F4, 16#62F6, 16#62F7, 16#62FC, 16#62FD, 16#62FE, 16#62FF, 16#6301, 16#6302, 16#6307, 16#6308, 16#6309, 16#630E, 16#6311, 16#6316, 16#631A, 16#631B, 16#631D, 16#631E, 16#631F, 16#6320, 16#6321, 16#6322, 16#6323, 16#6324, 16#6325, 16#6328, 16#632A, 16#632B, 16#632F, 16#6332, 16#6339, 16#633A, 16#633D, 16#6342, 16#6343, 16#6345, 16#6346, 16#6349, 16#634B, 16#634C, 16#634D, 16#634E, 16#634F, 16#6350, 16#6355, 16#635E, 16#635F, 16#6361, 16#6362, 16#6363, 16#6367, 16#6369, 16#636D, 16#636E, 16#6371, 16#6376, 16#6377, 16#637A, 16#637B, 16#6380, 16#6382, 16#6387, 16#6388, 16#6389, 16#638A, 16#638C, 16#638E, 16#638F, 16#6390, 16#6392, 16#6396, 16#6398, 16#63A0, 16#63A2, 16#63A3, 16#63A5, 16#63A7, 16#63A8, 16#63A9, 16#63AA, 16#63AC, 16#63AD, 16#63AE, 16#63B0, 16#63B3, 16#63B4, 16#63B7, 16#63B8, 16#63BA, 16#63BC, 16#63BE, 16#63C4, 16#63C6, 16#63C9, 16#63CD, 16#63CE, 16#63CF, 16#63D0, 16#63D2, 16#63D6, 16#63DE, 16#63E0, 16#63E1, 16#63E3, 16#63E9, 16#63EA, 16#63ED, 16#63F2, 16#63F4, 16#63F6, 16#63F8, 16#63FD, 16#63FF, 16#6400, 16#6401, 16#6402, 16#6405, 16#640B, 16#640C, 16#640F, 16#6410, 16#6413, 16#6414, 16#641B, 16#641C, 16#641E, 16#6420, 16#6421, 16#6426, 16#642A, 16#642C, 16#642D, 16#6434, 16#643A, 16#643D, 16#643F, 16#6441, 16#6444, 16#6445, 16#6446, 16#6447, 16#6448, 16#644A, 16#6452, 16#6454, 16#6458, 16#645E, 16#6467, 16#6469, 16#646D, 16#6478, 16#6479, 16#647A, 16#6482, 16#6484, 16#6485, 16#6487, 16#6491, 16#6492, 16#6495, 16#6496, 16#6499, 16#649E, 16#64A4, 16#64A9, 16#64AC, 16#64AD, 16#64AE, 16#64B0, 16#64B5, 16#64B7, 16#64B8, 16#64BA, 16#64BC, 16#64C0, 16#64C2, 16#64C5, 16#64CD, 16#64CE, 16#64D0, 16#64D2, 16#64D7, 16#64D8, 16#64DE, 16#64E2, 16#64E4, 16#64E6, 16#6500, 16#6509, 16#6512, 16#6518, 16#6525, 16#652B, 16#652E, 16#652F, 16#6534, 16#6535, 16#6536, 16#6538, 16#6539, 16#653B, 16#653E, 16#653F, 16#6545, 16#6548, 16#6549, 16#654C, 16#654F, 16#6551, 16#6555, 16#6556, 16#6559, 16#655B, 16#655D, 16#655E, 16#6562, 16#6563, 16#6566, 16#656B, 16#656C, 16#6570, 16#6572, 16#6574, 16#6577, 16#6587, 16#658B, 16#658C, 16#6590, 16#6591, 16#6593, 16#6597, 16#6599, 16#659B, 16#659C, 16#659F, 16#65A1, 16#65A4, 16#65A5, 16#65A7, 16#65A9, 16#65AB, 16#65AD, 16#65AF, 16#65B0, 16#65B9, 16#65BC, 16#65BD, 16#65C1, 16#65C3, 16#65C4, 16#65C5, 16#65C6, 16#65CB, 16#65CC, 16#65CE, 16#65CF, 16#65D2, 16#65D6, 16#65D7, 16#65E0, 16#65E2, 16#65E5, 16#65E6, 16#65E7, 16#65E8, 16#65E9, 16#65EC, 16#65ED, 16#65EE, 16#65EF, 16#65F0, 16#65F1, 16#65F6, 16#65F7, 16#65FA, 16#6600, 16#6602, 16#6603, 16#6606, 16#660A, 16#660C, 16#660E, 16#660F, 16#6613, 16#6614, 16#6615, 16#6619, 16#661D, 16#661F, 16#6620, 16#6625, 16#6627, 16#6628, 16#662D, 16#662F, 16#6631, 16#6634, 16#6635, 16#6636, 16#663C, 16#663E, 16#6641, 16#6643, 16#664B, 16#664C, 16#664F, 16#6652, 16#6653, 16#6654, 16#6655, 16#6656, 16#6657, 16#665A, 16#665F, 16#6661, 16#6664, 16#6666, 16#6668, 16#666E, 16#666F, 16#6670, 16#6674, 16#6676, 16#6677, 16#667A, 16#667E, 16#6682, 16#6684, 16#6687, 16#668C, 16#6691, 16#6696, 16#6697, 16#669D, 16#66A7, 16#66A8, 16#66AE, 16#66B4, 16#66B9, 16#66BE, 16#66D9, 16#66DB, 16#66DC, 16#66DD, 16#66E6, 16#66E9, 16#66F0, 16#66F2, 16#66F3, 16#66F4, 16#66F7, 16#66F9, 16#66FC, 16#66FE, 16#66FF, 16#6700, 16#6708, 16#6709, 16#670A, 16#670B, 16#670D, 16#6710, 16#6714, 16#6715, 16#6717, 16#671B, 16#671D, 16#671F, 16#6726, 16#6728, 16#672A, 16#672B, 16#672C, 16#672D, 16#672F, 16#6731, 16#6734, 16#6735, 16#673A, 16#673D, 16#6740, 16#6742, 16#6743, 16#6746, 16#6748, 16#6749, 16#674C, 16#674E, 16#674F, 16#6750, 16#6751, 16#6753, 16#6756, 16#675C, 16#675E, 16#675F, 16#6760, 16#6761, 16#6765, 16#6768, 16#6769, 16#676A, 16#676D, 16#676F, 16#6770, 16#6772, 16#6773, 16#6775, 16#6777, 16#677C, 16#677E, 16#677F, 16#6781, 16#6784, 16#6787, 16#6789, 16#678B, 16#6790, 16#6795, 16#6797, 16#6798, 16#679A, 16#679C, 16#679D, 16#679E, 16#67A2, 16#67A3, 16#67A5, 16#67A7, 16#67A8, 16#67AA, 16#67AB, 16#67AD, 16#67AF, 16#67B0, 16#67B3, 16#67B5, 16#67B6, 16#67B7, 16#67B8, 16#67C1, 16#67C3, 16#67C4, 16#67CF, 16#67D0, 16#67D1, 16#67D2, 16#67D3, 16#67D4, 16#67D8, 16#67D9, 16#67DA, 16#67DC, 16#67DD, 16#67DE, 16#67E0, 16#67E2, 16#67E5, 16#67E9, 16#67EC, 16#67EF, 16#67F0, 16#67F1, 16#67F3, 16#67F4, 16#67FD, 16#67FF, 16#6800, 16#6805, 16#6807, 16#6808, 16#6809, 16#680A, 16#680B, 16#680C, 16#680E, 16#680F, 16#6811, 16#6813, 16#6816, 16#6817, 16#681D, 16#6821, 16#6829, 16#682A, 16#6832, 16#6833, 16#6837, 16#6838, 16#6839, 16#683C, 16#683D, 16#683E, 16#6840, 16#6841, 16#6842, 16#6843, 16#6844, 16#6845, 16#6846, 16#6848, 16#6849, 16#684A, 16#684C, 16#684E, 16#6850, 16#6851, 16#6853, 16#6854, 16#6855, 16#6860, 16#6861, 16#6862, 16#6863, 16#6864, 16#6865, 16#6866, 16#6867, 16#6868, 16#6869, 16#686B, 16#6874, 16#6876, 16#6877, 16#6881, 16#6883, 16#6885, 16#6886, 16#688F, 16#6893, 16#6897, 16#68A2, 16#68A6, 16#68A7, 16#68A8, 16#68AD, 16#68AF, 16#68B0, 16#68B3, 16#68B5, 16#68C0, 16#68C2, 16#68C9, 16#68CB, 16#68CD, 16#68D2, 16#68D5, 16#68D8, 16#68DA, 16#68E0, 16#68E3, 16#68EE, 16#68F0, 16#68F1, 16#68F5, 16#68F9, 16#68FA, 16#68FC, 16#6901, 16#6905, 16#690B, 16#690D, 16#690E, 16#6910, 16#6912, 16#691F, 16#6920, 16#6924, 16#692D, 16#6930, 16#6934, 16#6939, 16#693D, 16#693F, 16#6942, 16#6954, 16#6957, 16#695A, 16#695D, 16#695E, 16#6960, 16#6963, 16#6966, 16#696B, 16#696E, 16#6971, 16#6977, 16#6978, 16#6979, 16#697C, 16#6980, 16#6982, 16#6984, 16#6986, 16#6987, 16#6988, 16#6989, 16#698D, 16#6994, 16#6995, 16#6998, 16#699B, 16#699C, 16#69A7, 16#69A8, 16#69AB, 16#69AD, 16#69B1, 16#69B4, 16#69B7, 16#69BB, 16#69C1, 16#69CA, 16#69CC, 16#69CE, 16#69D0, 16#69D4, 16#69DB, 16#69DF, 16#69E0, 16#69ED, 16#69F2, 16#69FD, 16#69FF, 16#6A0A, 16#6A17, 16#6A18, 16#6A1F, 16#6A21, 16#6A28, 16#6A2A, 16#6A2F, 16#6A31, 16#6A35, 16#6A3D, 16#6A3E, 16#6A44, 16#6A47, 16#6A50, 16#6A58, 16#6A59, 16#6A5B, 16#6A61, 16#6A65, 16#6A71, 16#6A79, 16#6A7C, 16#6A80, 16#6A84, 16#6A8E, 16#6A90, 16#6A91, 16#6A97, 16#6AA0, 16#6AA9, 16#6AAB, 16#6AAC, 16#6B20, 16#6B21, 16#6B22, 16#6B23, 16#6B24, 16#6B27, 16#6B32, 16#6B37, 16#6B39, 16#6B3A, 16#6B3E, 16#6B43, 16#6B46, 16#6B47, 16#6B49, 16#6B4C, 16#6B59, 16#6B62, 16#6B63, 16#6B64, 16#6B65, 16#6B66, 16#6B67, 16#6B6A, 16#6B79, 16#6B7B, 16#6B7C, 16#6B81, 16#6B82, 16#6B83, 16#6B84, 16#6B86, 16#6B87, 16#6B89, 16#6B8A, 16#6B8B, 16#6B8D, 16#6B92, 16#6B93, 16#6B96, 16#6B9A, 16#6B9B, 16#6BA1, 16#6BAA, 16#6BB3, 16#6BB4, 16#6BB5, 16#6BB7, 16#6BBF, 16#6BC1, 16#6BC2, 16#6BC5, 16#6BCB, 16#6BCD, 16#6BCF, 16#6BD2, 16#6BD3, 16#6BD4, 16#6BD5, 16#6BD6, 16#6BD7, 16#6BD9, 16#6BDB, 16#6BE1, 16#6BEA, 16#6BEB, 16#6BEF, 16#6BF3, 16#6BF5, 16#6BF9, 16#6BFD, 16#6C05, 16#6C06, 16#6C07, 16#6C0D, 16#6C0F, 16#6C10, 16#6C11, 16#6C13, 16#6C14, 16#6C15, 16#6C16, 16#6C18, 16#6C19, 16#6C1A, 16#6C1B, 16#6C1F, 16#6C21, 16#6C22, 16#6C24, 16#6C26, 16#6C27, 16#6C28, 16#6C29, 16#6C2A, 16#6C2E, 16#6C2F, 16#6C30, 16#6C32, 16#6C34, 16#6C35, 16#6C38, 16#6C3D, 16#6C40, 16#6C41, 16#6C42, 16#6C46, 16#6C47, 16#6C49, 16#6C4A, 16#6C50, 16#6C54, 16#6C55, 16#6C57, 16#6C5B, 16#6C5C, 16#6C5D, 16#6C5E, 16#6C5F, 16#6C60, 16#6C61, 16#6C64, 16#6C68, 16#6C69, 16#6C6A, 16#6C70, 16#6C72, 16#6C74, 16#6C76, 16#6C79, 16#6C7D, 16#6C7E, 16#6C81, 16#6C82, 16#6C83, 16#6C85, 16#6C86, 16#6C88, 16#6C89, 16#6C8C, 16#6C8F, 16#6C90, 16#6C93, 16#6C94, 16#6C99, 16#6C9B, 16#6C9F, 16#6CA1, 16#6CA3, 16#6CA4, 16#6CA5, 16#6CA6, 16#6CA7, 16#6CA9, 16#6CAA, 16#6CAB, 16#6CAD, 16#6CAE, 16#6CB1, 16#6CB2, 16#6CB3, 16#6CB8, 16#6CB9, 16#6CBB, 16#6CBC, 16#6CBD, 16#6CBE, 16#6CBF, 16#6CC4, 16#6CC5, 16#6CC9, 16#6CCA, 16#6CCC, 16#6CD0, 16#6CD3, 16#6CD4, 16#6CD5, 16#6CD6, 16#6CD7, 16#6CDB, 16#6CDE, 16#6CE0, 16#6CE1, 16#6CE2, 16#6CE3, 16#6CE5, 16#6CE8, 16#6CEA, 16#6CEB, 16#6CEE, 16#6CEF, 16#6CF0, 16#6CF1, 16#6CF3, 16#6CF5, 16#6CF6, 16#6CF7, 16#6CF8, 16#6CFA, 16#6CFB, 16#6CFC, 16#6CFD, 16#6CFE, 16#6D01, 16#6D04, 16#6D07, 16#6D0B, 16#6D0C, 16#6D0E, 16#6D12, 16#6D17, 16#6D19, 16#6D1A, 16#6D1B, 16#6D1E, 16#6D25, 16#6D27, 16#6D2A, 16#6D2B, 16#6D2E, 16#6D31, 16#6D32, 16#6D33, 16#6D35, 16#6D39, 16#6D3B, 16#6D3C, 16#6D3D, 16#6D3E, 16#6D41, 16#6D43, 16#6D45, 16#6D46, 16#6D47, 16#6D48, 16#6D4A, 16#6D4B, 16#6D4D, 16#6D4E, 16#6D4F, 16#6D51, 16#6D52, 16#6D53, 16#6D54, 16#6D59, 16#6D5A, 16#6D5C, 16#6D5E, 16#6D60, 16#6D63, 16#6D66, 16#6D69, 16#6D6A, 16#6D6E, 16#6D6F, 16#6D74, 16#6D77, 16#6D78, 16#6D7C, 16#6D82, 16#6D85, 16#6D88, 16#6D89, 16#6D8C, 16#6D8E, 16#6D91, 16#6D93, 16#6D94, 16#6D95, 16#6D9B, 16#6D9D, 16#6D9E, 16#6D9F, 16#6DA0, 16#6DA1, 16#6DA3, 16#6DA4, 16#6DA6, 16#6DA7, 16#6DA8, 16#6DA9, 16#6DAA, 16#6DAB, 16#6DAE, 16#6DAF, 16#6DB2, 16#6DB5, 16#6DB8, 16#6DBF, 16#6DC0, 16#6DC4, 16#6DC5, 16#6DC6, 16#6DC7, 16#6DCB, 16#6DCC, 16#6DD1, 16#6DD6, 16#6DD8, 16#6DD9, 16#6DDD, 16#6DDE, 16#6DE0, 16#6DE1, 16#6DE4, 16#6DE6, 16#6DEB, 16#6DEC, 16#6DEE, 16#6DF1, 16#6DF3, 16#6DF7, 16#6DF9, 16#6DFB, 16#6DFC, 16#6E05, 16#6E0A, 16#6E0C, 16#6E0D, 16#6E0E, 16#6E10, 16#6E11, 16#6E14, 16#6E16, 16#6E17, 16#6E1A, 16#6E1D, 16#6E20, 16#6E21, 16#6E23, 16#6E24, 16#6E25, 16#6E29, 16#6E2B, 16#6E2D, 16#6E2F, 16#6E32, 16#6E34, 16#6E38, 16#6E3A, 16#6E43, 16#6E44, 16#6E4D, 16#6E4E, 16#6E53, 16#6E54, 16#6E56, 16#6E58, 16#6E5B, 16#6E5F, 16#6E6B, 16#6E6E, 16#6E7E, 16#6E7F, 16#6E83, 16#6E85, 16#6E86, 16#6E89, 16#6E8F, 16#6E90, 16#6E98, 16#6E9C, 16#6E9F, 16#6EA2, 16#6EA5, 16#6EA7, 16#6EAA, 16#6EAF, 16#6EB1, 16#6EB2, 16#6EB4, 16#6EB6, 16#6EB7, 16#6EBA, 16#6EBB, 16#6EBD, 16#6EC1, 16#6EC2, 16#6EC7, 16#6ECB, 16#6ECF, 16#6ED1, 16#6ED3, 16#6ED4, 16#6ED5, 16#6ED7, 16#6EDA, 16#6EDE, 16#6EDF, 16#6EE0, 16#6EE1, 16#6EE2, 16#6EE4, 16#6EE5, 16#6EE6, 16#6EE8, 16#6EE9, 16#6EF4, 16#6EF9, 16#6F02, 16#6F06, 16#6F09, 16#6F0F, 16#6F13, 16#6F14, 16#6F15, 16#6F20, 16#6F24, 16#6F29, 16#6F2A, 16#6F2B, 16#6F2D, 16#6F2F, 16#6F31, 16#6F33, 16#6F36, 16#6F3E, 16#6F46, 16#6F47, 16#6F4B, 16#6F4D, 16#6F58, 16#6F5C, 16#6F5E, 16#6F62, 16#6F66, 16#6F6D, 16#6F6E, 16#6F72, 16#6F74, 16#6F78, 16#6F7A, 16#6F7C, 16#6F84, 16#6F88, 16#6F89, 16#6F8C, 16#6F8D, 16#6F8E, 16#6F9C, 16#6FA1, 16#6FA7, 16#6FB3, 16#6FB6, 16#6FB9, 16#6FC0, 16#6FC2, 16#6FC9, 16#6FD1, 16#6FD2, 16#6FDE, 16#6FE0, 16#6FE1, 16#6FEE, 16#6FEF, 16#7011, 16#701A, 16#701B, 16#7023, 16#7035, 16#7039, 16#704C, 16#704F, 16#705E, 16#706B, 16#706C, 16#706D, 16#706F, 16#7070, 16#7075, 16#7076, 16#7078, 16#707C, 16#707E, 16#707F, 16#7080, 16#7085, 16#7089, 16#708A, 16#708E, 16#7092, 16#7094, 16#7095, 16#7096, 16#7099, 16#709C, 16#709D, 16#70AB, 16#70AC, 16#70AD, 16#70AE, 16#70AF, 16#70B1, 16#70B3, 16#70B7, 16#70B8, 16#70B9, 16#70BB, 16#70BC, 16#70BD, 16#70C0, 16#70C1, 16#70C2, 16#70C3, 16#70C8, 16#70CA, 16#70D8, 16#70D9, 16#70DB, 16#70DF, 16#70E4, 16#70E6, 16#70E7, 16#70E8, 16#70E9, 16#70EB, 16#70EC, 16#70ED, 16#70EF, 16#70F7, 16#70F9, 16#70FD, 16#7109, 16#710A, 16#7110, 16#7113, 16#7115, 16#7116, 16#7118, 16#7119, 16#711A, 16#7126, 16#712F, 16#7130, 16#7131, 16#7136, 16#7145, 16#714A, 16#714C, 16#714E, 16#715C, 16#715E, 16#7164, 16#7166, 16#7167, 16#7168, 16#716E, 16#7172, 16#7173, 16#7178, 16#717A, 16#717D, 16#7184, 16#718A, 16#718F, 16#7194, 16#7198, 16#7199, 16#719F, 16#71A0, 16#71A8, 16#71AC, 16#71B3, 16#71B5, 16#71B9, 16#71C3, 16#71CE, 16#71D4, 16#71D5, 16#71E0, 16#71E5, 16#71E7, 16#71EE, 16#71F9, 16#7206, 16#721D, 16#7228, 16#722A, 16#722C, 16#7230, 16#7231, 16#7235, 16#7236, 16#7237, 16#7238, 16#7239, 16#723B, 16#723D, 16#723F, 16#7247, 16#7248, 16#724C, 16#724D, 16#7252, 16#7256, 16#7259, 16#725B, 16#725D, 16#725F, 16#7261, 16#7262, 16#7266, 16#7267, 16#7269, 16#726E, 16#726F, 16#7272, 16#7275, 16#7279, 16#727A, 16#727E, 16#727F, 16#7280, 16#7281, 16#7284, 16#728A, 16#728B, 16#728D, 16#728F, 16#7292, 16#729F, 16#72AC, 16#72AD, 16#72AF, 16#72B0, 16#72B4, 16#72B6, 16#72B7, 16#72B8, 16#72B9, 16#72C1, 16#72C2, 16#72C3, 16#72C4, 16#72C8, 16#72CD, 16#72CE, 16#72D0, 16#72D2, 16#72D7, 16#72D9, 16#72DE, 16#72E0, 16#72E1, 16#72E8, 16#72E9, 16#72EC, 16#72ED, 16#72EE, 16#72EF, 16#72F0, 16#72F1, 16#72F2, 16#72F3, 16#72F4, 16#72F7, 16#72F8, 16#72FA, 16#72FB, 16#72FC, 16#7301, 16#7303, 16#730A, 16#730E, 16#7313, 16#7315, 16#7316, 16#7317, 16#731B, 16#731C, 16#731D, 16#731E, 16#7321, 16#7322, 16#7325, 16#7329, 16#732A, 16#732B, 16#732C, 16#732E, 16#7331, 16#7334, 16#7337, 16#7338, 16#7339, 16#733E, 16#733F, 16#734D, 16#7350, 16#7352, 16#7357, 16#7360, 16#736C, 16#736D, 16#736F, 16#737E, 16#7384, 16#7387, 16#7389, 16#738B, 16#738E, 16#7391, 16#7396, 16#739B, 16#739F, 16#73A2, 16#73A9, 16#73AB, 16#73AE, 16#73AF, 16#73B0, 16#73B2, 16#73B3, 16#73B7, 16#73BA, 16#73BB, 16#73C0, 16#73C2, 16#73C8, 16#73C9, 16#73CA, 16#73CD, 16#73CF, 16#73D0, 16#73D1, 16#73D9, 16#73DE, 16#73E0, 16#73E5, 16#73E7, 16#73E9, 16#73ED, 16#73F2, 16#7403, 16#7405, 16#7406, 16#7409, 16#740A, 16#740F, 16#7410, 16#741A, 16#741B, 16#7422, 16#7425, 16#7426, 16#7428, 16#742A, 16#742C, 16#742E, 16#7430, 16#7433, 16#7434, 16#7435, 16#7436, 16#743C, 16#7441, 16#7455, 16#7457, 16#7459, 16#745A, 16#745B, 16#745C, 16#745E, 16#745F, 16#746D, 16#7470, 16#7476, 16#7477, 16#747E, 16#7480, 16#7481, 16#7483, 16#7487, 16#748B, 16#748E, 16#7490, 16#749C, 16#749E, 16#74A7, 16#74A8, 16#74A9, 16#74BA, 16#74D2, 16#74DC, 16#74DE, 16#74E0, 16#74E2, 16#74E3, 16#74E4, 16#74E6, 16#74EE, 16#74EF, 16#74F4, 16#74F6, 16#74F7, 16#74FF, 16#7504, 16#750D, 16#750F, 16#7511, 16#7513, 16#7518, 16#7519, 16#751A, 16#751C, 16#751F, 16#7525, 16#7528, 16#7529, 16#752B, 16#752C, 16#752D, 16#752F, 16#7530, 16#7531, 16#7532, 16#7533, 16#7535, 16#7537, 16#7538, 16#753A, 16#753B, 16#753E, 16#7540, 16#7545, 16#7548, 16#754B, 16#754C, 16#754E, 16#754F, 16#7554, 16#7559, 16#755A, 16#755B, 16#755C, 16#7565, 16#7566, 16#756A, 16#7572, 16#7574, 16#7578, 16#7579, 16#757F, 16#7583, 16#7586, 16#758B, 16#758F, 16#7591, 16#7592, 16#7594, 16#7596, 16#7597, 16#7599, 16#759A, 16#759D, 16#759F, 16#75A0, 16#75A1, 16#75A3, 16#75A4, 16#75A5, 16#75AB, 16#75AC, 16#75AE, 16#75AF, 16#75B0, 16#75B1, 16#75B2, 16#75B3, 16#75B4, 16#75B5, 16#75B8, 16#75B9, 16#75BC, 16#75BD, 16#75BE, 16#75C2, 16#75C3, 16#75C4, 16#75C5, 16#75C7, 16#75C8, 16#75C9, 16#75CA, 16#75CD, 16#75D2, 16#75D4, 16#75D5, 16#75D6, 16#75D8, 16#75DB, 16#75DE, 16#75E2, 16#75E3, 16#75E4, 16#75E6, 16#75E7, 16#75E8, 16#75EA, 16#75EB, 16#75F0, 16#75F1, 16#75F4, 16#75F9, 16#75FC, 16#75FF, 16#7600, 16#7601, 16#7603, 16#7605, 16#760A, 16#760C, 16#7610, 16#7615, 16#7617, 16#7618, 16#7619, 16#761B, 16#761F, 16#7620, 16#7622, 16#7624, 16#7625, 16#7626, 16#7629, 16#762A, 16#762B, 16#762D, 16#7630, 16#7633, 16#7634, 16#7635, 16#7638, 16#763C, 16#763E, 16#763F, 16#7640, 16#7643, 16#764C, 16#764D, 16#7654, 16#7656, 16#765C, 16#765E, 16#7663, 16#766B, 16#766F, 16#7678, 16#767B, 16#767D, 16#767E, 16#7682, 16#7684, 16#7686, 16#7687, 16#7688, 16#768B, 16#768E, 16#7691, 16#7693, 16#7696, 16#7699, 16#76A4, 16#76AE, 16#76B1, 16#76B2, 16#76B4, 16#76BF, 16#76C2, 16#76C5, 16#76C6, 16#76C8, 16#76CA, 16#76CD, 16#76CE, 16#76CF, 16#76D0, 16#76D1, 16#76D2, 16#76D4, 16#76D6, 16#76D7, 16#76D8, 16#76DB, 16#76DF, 16#76E5, 16#76EE, 16#76EF, 16#76F1, 16#76F2, 16#76F4, 16#76F8, 16#76F9, 16#76FC, 16#76FE, 16#7701, 16#7704, 16#7707, 16#7708, 16#7709, 16#770B, 16#770D, 16#7719, 16#771A, 16#771F, 16#7720, 16#7722, 16#7726, 16#7728, 16#7729, 16#772D, 16#772F, 16#7735, 16#7736, 16#7737, 16#7738, 16#773A, 16#773C, 16#7740, 16#7741, 16#7743, 16#7747, 16#7750, 16#7751, 16#775A, 16#775B, 16#7761, 16#7762, 16#7763, 16#7765, 16#7766, 16#7768, 16#776B, 16#776C, 16#7779, 16#777D, 16#777E, 16#777F, 16#7780, 16#7784, 16#7785, 16#778C, 16#778D, 16#778E, 16#7791, 16#7792, 16#779F, 16#77A0, 16#77A2, 16#77A5, 16#77A7, 16#77A9, 16#77AA, 16#77AC, 16#77B0, 16#77B3, 16#77B5, 16#77BB, 16#77BD, 16#77BF, 16#77CD, 16#77D7, 16#77DB, 16#77DC, 16#77E2, 16#77E3, 16#77E5, 16#77E7, 16#77E9, 16#77EB, 16#77EC, 16#77ED, 16#77EE, 16#77F3, 16#77F6, 16#77F8, 16#77FD, 16#77FE, 16#77FF, 16#7800, 16#7801, 16#7802, 16#7809, 16#780C, 16#780D, 16#7811, 16#7812, 16#7814, 16#7816, 16#7817, 16#7818, 16#781A, 16#781C, 16#781D, 16#781F, 16#7823, 16#7825, 16#7826, 16#7827, 16#7829, 16#782C, 16#782D, 16#7830, 16#7834, 16#7837, 16#7838, 16#7839, 16#783A, 16#783B, 16#783C, 16#783E, 16#7840, 16#7845, 16#7847, 16#784C, 16#784E, 16#7850, 16#7852, 16#7855, 16#7856, 16#7857, 16#785D, 16#786A, 16#786B, 16#786C, 16#786D, 16#786E, 16#7877, 16#787C, 16#7887, 16#7889, 16#788C, 16#788D, 16#788E, 16#7891, 16#7893, 16#7897, 16#7898, 16#789A, 16#789B, 16#789C, 16#789F, 16#78A1, 16#78A3, 16#78A5, 16#78A7, 16#78B0, 16#78B1, 16#78B2, 16#78B3, 16#78B4, 16#78B9, 16#78BE, 16#78C1, 16#78C5, 16#78C9, 16#78CA, 16#78CB, 16#78D0, 16#78D4, 16#78D5, 16#78D9, 16#78E8, 16#78EC, 16#78F2, 16#78F4, 16#78F7, 16#78FA, 16#7901, 16#7905, 16#7913, 16#791E, 16#7924, 16#7934, 16#793A, 16#793B, 16#793C, 16#793E, 16#7940, 16#7941, 16#7946, 16#7948, 16#7949, 16#7953, 16#7956, 16#7957, 16#795A, 16#795B, 16#795C, 16#795D, 16#795E, 16#795F, 16#7960, 16#7962, 16#7965, 16#7967, 16#7968, 16#796D, 16#796F, 16#7977, 16#7978, 16#797A, 16#7980, 16#7981, 16#7984, 16#7985, 16#798A, 16#798F, 16#799A, 16#79A7, 16#79B3, 16#79B9, 16#79BA, 16#79BB, 16#79BD, 16#79BE, 16#79C0, 16#79C1, 16#79C3, 16#79C6, 16#79C9, 16#79CB, 16#79CD, 16#79D1, 16#79D2, 16#79D5, 16#79D8, 16#79DF, 16#79E3, 16#79E4, 16#79E6, 16#79E7, 16#79E9, 16#79EB, 16#79ED, 16#79EF, 16#79F0, 16#79F8, 16#79FB, 16#79FD, 16#7A00, 16#7A02, 16#7A03, 16#7A06, 16#7A0B, 16#7A0D, 16#7A0E, 16#7A14, 16#7A17, 16#7A1A, 16#7A1E, 16#7A20, 16#7A23, 16#7A33, 16#7A37, 16#7A39, 16#7A3B, 16#7A3C, 16#7A3D, 16#7A3F, 16#7A46, 16#7A51, 16#7A57, 16#7A70, 16#7A74, 16#7A76, 16#7A77, 16#7A78, 16#7A79, 16#7A7A, 16#7A7F, 16#7A80, 16#7A81, 16#7A83, 16#7A84, 16#7A86, 16#7A88, 16#7A8D, 16#7A91, 16#7A92, 16#7A95, 16#7A96, 16#7A97, 16#7A98, 16#7A9C, 16#7A9D, 16#7A9F, 16#7AA0, 16#7AA5, 16#7AA6, 16#7AA8, 16#7AAC, 16#7AAD, 16#7AB3, 16#7ABF, 16#7ACB, 16#7AD6, 16#7AD9, 16#7ADE, 16#7ADF, 16#7AE0, 16#7AE3, 16#7AE5, 16#7AE6, 16#7AED, 16#7AEF, 16#7AF9, 16#7AFA, 16#7AFD, 16#7AFF, 16#7B03, 16#7B04, 16#7B06, 16#7B08, 16#7B0A, 16#7B0B, 16#7B0F, 16#7B11, 16#7B14, 16#7B15, 16#7B19, 16#7B1B, 16#7B1E, 16#7B20, 16#7B24, 16#7B25, 16#7B26, 16#7B28, 16#7B2A, 16#7B2B, 16#7B2C, 16#7B2E, 16#7B31, 16#7B33, 16#7B38, 16#7B3A, 16#7B3C, 16#7B3E, 16#7B45, 16#7B47, 16#7B49, 16#7B4B, 16#7B4C, 16#7B4F, 16#7B50, 16#7B51, 16#7B52, 16#7B54, 16#7B56, 16#7B58, 16#7B5A, 16#7B5B, 16#7B5D, 16#7B60, 16#7B62, 16#7B6E, 16#7B71, 16#7B72, 16#7B75, 16#7B77, 16#7B79, 16#7B7B, 16#7B7E, 16#7B80, 16#7B85, 16#7B8D, 16#7B90, 16#7B94, 16#7B95, 16#7B97, 16#7B9C, 16#7B9D, 16#7BA1, 16#7BA2, 16#7BA6, 16#7BA7, 16#7BA8, 16#7BA9, 16#7BAA, 16#7BAB, 16#7BAC, 16#7BAD, 16#7BB1, 16#7BB4, 16#7BB8, 16#7BC1, 16#7BC6, 16#7BC7, 16#7BCC, 16#7BD1, 16#7BD3, 16#7BD9, 16#7BDA, 16#7BDD, 16#7BE1, 16#7BE5, 16#7BE6, 16#7BEA, 16#7BEE, 16#7BF1, 16#7BF7, 16#7BFC, 16#7BFE, 16#7C07, 16#7C0B, 16#7C0C, 16#7C0F, 16#7C16, 16#7C1F, 16#7C26, 16#7C27, 16#7C2A, 16#7C38, 16#7C3F, 16#7C40, 16#7C41, 16#7C4D, 16#7C73, 16#7C74, 16#7C7B, 16#7C7C, 16#7C7D, 16#7C89, 16#7C91, 16#7C92, 16#7C95, 16#7C97, 16#7C98, 16#7C9C, 16#7C9D, 16#7C9E, 16#7C9F, 16#7CA2, 16#7CA4, 16#7CA5, 16#7CAA, 16#7CAE, 16#7CB1, 16#7CB2, 16#7CB3, 16#7CB9, 16#7CBC, 16#7CBD, 16#7CBE, 16#7CC1, 16#7CC5, 16#7CC7, 16#7CC8, 16#7CCA, 16#7CCC, 16#7CCD, 16#7CD5, 16#7CD6, 16#7CD7, 16#7CD9, 16#7CDC, 16#7CDF, 16#7CE0, 16#7CE8, 16#7CEF, 16#7CF8, 16#7CFB, 16#7D0A, 16#7D20, 16#7D22, 16#7D27, 16#7D2B, 16#7D2F, 16#7D6E, 16#7D77, 16#7DA6, 16#7DAE, 16#7E3B, 16#7E41, 16#7E47, 16#7E82, 16#7E9B, 16#7E9F, 16#7EA0, 16#7EA1, 16#7EA2, 16#7EA3, 16#7EA4, 16#7EA5, 16#7EA6, 16#7EA7, 16#7EA8, 16#7EA9, 16#7EAA, 16#7EAB, 16#7EAC, 16#7EAD, 16#7EAF, 16#7EB0, 16#7EB1, 16#7EB2, 16#7EB3, 16#7EB5, 16#7EB6, 16#7EB7, 16#7EB8, 16#7EB9, 16#7EBA, 16#7EBD, 16#7EBE, 16#7EBF, 16#7EC0, 16#7EC1, 16#7EC2, 16#7EC3, 16#7EC4, 16#7EC5, 16#7EC6, 16#7EC7, 16#7EC8, 16#7EC9, 16#7ECA, 16#7ECB, 16#7ECC, 16#7ECD, 16#7ECE, 16#7ECF, 16#7ED0, 16#7ED1, 16#7ED2, 16#7ED3, 16#7ED4, 16#7ED5, 16#7ED7, 16#7ED8, 16#7ED9, 16#7EDA, 16#7EDB, 16#7EDC, 16#7EDD, 16#7EDE, 16#7EDF, 16#7EE0, 16#7EE1, 16#7EE2, 16#7EE3, 16#7EE5, 16#7EE6, 16#7EE7, 16#7EE8, 16#7EE9, 16#7EEA, 16#7EEB, 16#7EED, 16#7EEE, 16#7EEF, 16#7EF0, 16#7EF1, 16#7EF2, 16#7EF3, 16#7EF4, 16#7EF5, 16#7EF6, 16#7EF7, 16#7EF8, 16#7EFA, 16#7EFB, 16#7EFC, 16#7EFD, 16#7EFE, 16#7EFF, 16#7F00, 16#7F01, 16#7F02, 16#7F03, 16#7F04, 16#7F05, 16#7F06, 16#7F07, 16#7F08, 16#7F09, 16#7F0B, 16#7F0C, 16#7F0D, 16#7F0E, 16#7F0F, 16#7F11, 16#7F12, 16#7F13, 16#7F14, 16#7F15, 16#7F16, 16#7F17, 16#7F18, 16#7F19, 16#7F1A, 16#7F1B, 16#7F1C, 16#7F1D, 16#7F1F, 16#7F20, 16#7F21, 16#7F22, 16#7F23, 16#7F24, 16#7F25, 16#7F26, 16#7F27, 16#7F28, 16#7F29, 16#7F2A, 16#7F2B, 16#7F2C, 16#7F2D, 16#7F2E, 16#7F2F, 16#7F30, 16#7F31, 16#7F32, 16#7F33, 16#7F34, 16#7F35, 16#7F36, 16#7F38, 16#7F3A, 16#7F42, 16#7F44, 16#7F45, 16#7F50, 16#7F51, 16#7F54, 16#7F55, 16#7F57, 16#7F58, 16#7F5A, 16#7F5F, 16#7F61, 16#7F62, 16#7F68, 16#7F69, 16#7F6A, 16#7F6E, 16#7F71, 16#7F72, 16#7F74, 16#7F79, 16#7F7E, 16#7F81, 16#7F8A, 16#7F8C, 16#7F8E, 16#7F94, 16#7F9A, 16#7F9D, 16#7F9E, 16#7F9F, 16#7FA1, 16#7FA4, 16#7FA7, 16#7FAF, 16#7FB0, 16#7FB2, 16#7FB8, 16#7FB9, 16#7FBC, 16#7FBD, 16#7FBF, 16#7FC1, 16#7FC5, 16#7FCA, 16#7FCC, 16#7FCE, 16#7FD4, 16#7FD5, 16#7FD8, 16#7FDF, 16#7FE0, 16#7FE1, 16#7FE5, 16#7FE6, 16#7FE9, 16#7FEE, 16#7FF0, 16#7FF1, 16#7FF3, 16#7FFB, 16#7FFC, 16#8000, 16#8001, 16#8003, 16#8004, 16#8005, 16#8006, 16#800B, 16#800C, 16#800D, 16#8010, 16#8012, 16#8014, 16#8015, 16#8016, 16#8017, 16#8018, 16#8019, 16#801C, 16#8020, 16#8022, 16#8025, 16#8026, 16#8027, 16#8028, 16#8029, 16#802A, 16#8031, 16#8033, 16#8035, 16#8036, 16#8037, 16#8038, 16#803B, 16#803D, 16#803F, 16#8042, 16#8043, 16#8046, 16#804A, 16#804B, 16#804C, 16#804D, 16#8052, 16#8054, 16#8058, 16#805A, 16#8069, 16#806A, 16#8071, 16#807F, 16#8080, 16#8083, 16#8084, 16#8086, 16#8087, 16#8089, 16#808B, 16#808C, 16#8093, 16#8096, 16#8098, 16#809A, 16#809B, 16#809C, 16#809D, 16#809F, 16#80A0, 16#80A1, 16#80A2, 16#80A4, 16#80A5, 16#80A9, 16#80AA, 16#80AB, 16#80AD, 16#80AE, 16#80AF, 16#80B1, 16#80B2, 16#80B4, 16#80B7, 16#80BA, 16#80BC, 16#80BD, 16#80BE, 16#80BF, 16#80C0, 16#80C1, 16#80C2, 16#80C3, 16#80C4, 16#80C6, 16#80CC, 16#80CD, 16#80CE, 16#80D6, 16#80D7, 16#80D9, 16#80DA, 16#80DB, 16#80DC, 16#80DD, 16#80DE, 16#80E1, 16#80E4, 16#80E5, 16#80E7, 16#80E8, 16#80E9, 16#80EA, 16#80EB, 16#80EC, 16#80ED, 16#80EF, 16#80F0, 16#80F1, 16#80F2, 16#80F3, 16#80F4, 16#80F6, 16#80F8, 16#80FA, 16#80FC, 16#80FD, 16#8102, 16#8106, 16#8109, 16#810A, 16#810D, 16#810E, 16#810F, 16#8110, 16#8111, 16#8112, 16#8113, 16#8114, 16#8116, 16#8118, 16#811A, 16#811E, 16#812C, 16#812F, 16#8131, 16#8132, 16#8136, 16#8138, 16#813E, 16#8146, 16#8148, 16#814A, 16#814B, 16#814C, 16#8150, 16#8151, 16#8153, 16#8154, 16#8155, 16#8159, 16#815A, 16#8160, 16#8165, 16#8167, 16#8169, 16#816D, 16#816E, 16#8170, 16#8171, 16#8174, 16#8179, 16#817A, 16#817B, 16#817C, 16#817D, 16#817E, 16#817F, 16#8180, 16#8182, 16#8188, 16#818A, 16#818F, 16#8191, 16#8198, 16#819B, 16#819C, 16#819D, 16#81A3, 16#81A6, 16#81A8, 16#81AA, 16#81B3, 16#81BA, 16#81BB, 16#81C0, 16#81C1, 16#81C2, 16#81C3, 16#81C6, 16#81CA, 16#81CC, 16#81E3, 16#81E7, 16#81EA, 16#81EC, 16#81ED, 16#81F3, 16#81F4, 16#81FB, 16#81FC, 16#81FE, 16#8200, 16#8201, 16#8202, 16#8204, 16#8205, 16#8206, 16#820C, 16#820D, 16#8210, 16#8212, 16#8214, 16#821B, 16#821C, 16#821E, 16#821F, 16#8221, 16#8222, 16#8223, 16#8228, 16#822A, 16#822B, 16#822C, 16#822D, 16#822F, 16#8230, 16#8231, 16#8233, 16#8234, 16#8235, 16#8236, 16#8237, 16#8238, 16#8239, 16#823B, 16#823E, 16#8244, 16#8247, 16#8249, 16#824B, 16#824F, 16#8258, 16#825A, 16#825F, 16#8268, 16#826E, 16#826F, 16#8270, 16#8272, 16#8273, 16#8274, 16#8279, 16#827A, 16#827D, 16#827E, 16#827F, 16#8282, 16#8284, 16#8288, 16#828A, 16#828B, 16#828D, 16#828E, 16#828F, 16#8291, 16#8292, 16#8297, 16#8298, 16#8299, 16#829C, 16#829D, 16#829F, 16#82A1, 16#82A4, 16#82A5, 16#82A6, 16#82A8, 16#82A9, 16#82AA, 16#82AB, 16#82AC, 16#82AD, 16#82AE, 16#82AF, 16#82B0, 16#82B1, 16#82B3, 16#82B4, 16#82B7, 16#82B8, 16#82B9, 16#82BD, 16#82BE, 16#82C1, 16#82C4, 16#82C7, 16#82C8, 16#82CA, 16#82CB, 16#82CC, 16#82CD, 16#82CE, 16#82CF, 16#82D1, 16#82D2, 16#82D3, 16#82D4, 16#82D5, 16#82D7, 16#82D8, 16#82DB, 16#82DC, 16#82DE, 16#82DF, 16#82E0, 16#82E1, 16#82E3, 16#82E4, 16#82E5, 16#82E6, 16#82EB, 16#82EF, 16#82F1, 16#82F4, 16#82F7, 16#82F9, 16#82FB, 16#8301, 16#8302, 16#8303, 16#8304, 16#8305, 16#8306, 16#8307, 16#8308, 16#8309, 16#830C, 16#830E, 16#830F, 16#8311, 16#8314, 16#8315, 16#8317, 16#831A, 16#831B, 16#831C, 16#8327, 16#8328, 16#832B, 16#832C, 16#832D, 16#832F, 16#8331, 16#8333, 16#8334, 16#8335, 16#8336, 16#8338, 16#8339, 16#833A, 16#833C, 16#8340, 16#8343, 16#8346, 16#8347, 16#8349, 16#834F, 16#8350, 16#8351, 16#8352, 16#8354, 16#835A, 16#835B, 16#835C, 16#835E, 16#835F, 16#8360, 16#8361, 16#8363, 16#8364, 16#8365, 16#8366, 16#8367, 16#8368, 16#8369, 16#836A, 16#836B, 16#836C, 16#836D, 16#836E, 16#836F, 16#8377, 16#8378, 16#837B, 16#837C, 16#837D, 16#8385, 16#8386, 16#8389, 16#838E, 16#8392, 16#8393, 16#8398, 16#839B, 16#839C, 16#839E, 16#83A0, 16#83A8, 16#83A9, 16#83AA, 16#83AB, 16#83B0, 16#83B1, 16#83B2, 16#83B3, 16#83B4, 16#83B6, 16#83B7, 16#83B8, 16#83B9, 16#83BA, 16#83BC, 16#83BD, 16#83C0, 16#83C1, 16#83C5, 16#83C7, 16#83CA, 16#83CC, 16#83CF, 16#83D4, 16#83D6, 16#83D8, 16#83DC, 16#83DD, 16#83DF, 16#83E0, 16#83E1, 16#83E5, 16#83E9, 16#83EA, 16#83F0, 16#83F1, 16#83F2, 16#83F8, 16#83F9, 16#83FD, 16#8401, 16#8403, 16#8404, 16#8406, 16#840B, 16#840C, 16#840D, 16#840E, 16#840F, 16#8411, 16#8418, 16#841C, 16#841D, 16#8424, 16#8425, 16#8426, 16#8427, 16#8428, 16#8431, 16#8438, 16#843C, 16#843D, 16#8446, 16#8451, 16#8457, 16#8459, 16#845A, 16#845B, 16#845C, 16#8461, 16#8463, 16#8469, 16#846B, 16#846C, 16#846D, 16#8471, 16#8473, 16#8475, 16#8476, 16#8478, 16#847A, 16#8482, 16#8487, 16#8488, 16#8489, 16#848B, 16#848C, 16#848E, 16#8497, 16#8499, 16#849C, 16#84A1, 16#84AF, 16#84B2, 16#84B4, 16#84B8, 16#84B9, 16#84BA, 16#84BD, 16#84BF, 16#84C1, 16#84C4, 16#84C9, 16#84CA, 16#84CD, 16#84D0, 16#84D1, 16#84D3, 16#84D6, 16#84DD, 16#84DF, 16#84E0, 16#84E3, 16#84E5, 16#84E6, 16#84EC, 16#84F0, 16#84FC, 16#84FF, 16#850C, 16#8511, 16#8513, 16#8517, 16#851A, 16#851F, 16#8521, 16#852B, 16#852C, 16#8537, 16#8538, 16#8539, 16#853A, 16#853B, 16#853C, 16#853D, 16#8543, 16#8548, 16#8549, 16#854A, 16#8556, 16#8559, 16#855E, 16#8564, 16#8568, 16#8572, 16#8574, 16#8579, 16#857A, 16#857B, 16#857E, 16#8584, 16#8585, 16#8587, 16#858F, 16#859B, 16#859C, 16#85A4, 16#85A8, 16#85AA, 16#85AE, 16#85AF, 16#85B0, 16#85B7, 16#85B9, 16#85C1, 16#85C9, 16#85CF, 16#85D0, 16#85D3, 16#85D5, 16#85DC, 16#85E4, 16#85E9, 16#85FB, 16#85FF, 16#8605, 16#8611, 16#8616, 16#8627, 16#8629, 16#8638, 16#863C, 16#864D, 16#864E, 16#864F, 16#8650, 16#8651, 16#8654, 16#865A, 16#865E, 16#8662, 16#866B, 16#866C, 16#866E, 16#8671, 16#8679, 16#867A, 16#867B, 16#867C, 16#867D, 16#867E, 16#867F, 16#8680, 16#8681, 16#8682, 16#868A, 16#868B, 16#868C, 16#868D, 16#8693, 16#8695, 16#869C, 16#869D, 16#86A3, 16#86A4, 16#86A7, 16#86A8, 16#86A9, 16#86AA, 16#86AC, 16#86AF, 16#86B0, 16#86B1, 16#86B4, 16#86B5, 16#86B6, 16#86BA, 16#86C0, 16#86C4, 16#86C6, 16#86C7, 16#86C9, 16#86CA, 16#86CB, 16#86CE, 16#86CF, 16#86D0, 16#86D1, 16#86D4, 16#86D8, 16#86D9, 16#86DB, 16#86DE, 16#86DF, 16#86E4, 16#86E9, 16#86ED, 16#86EE, 16#86F0, 16#86F1, 16#86F2, 16#86F3, 16#86F4, 16#86F8, 16#86F9, 16#86FE, 16#8700, 16#8702, 16#8703, 16#8707, 16#8708, 16#8709, 16#870A, 16#870D, 16#8712, 16#8713, 16#8715, 16#8717, 16#8718, 16#871A, 16#871C, 16#871E, 16#8721, 16#8722, 16#8723, 16#8725, 16#8729, 16#872E, 16#8731, 16#8734, 16#8737, 16#873B, 16#873E, 16#873F, 16#8747, 16#8748, 16#8749, 16#874C, 16#874E, 16#8753, 16#8757, 16#8759, 16#8760, 16#8763, 16#8764, 16#8765, 16#876E, 16#8770, 16#8774, 16#8776, 16#877B, 16#877C, 16#877D, 16#877E, 16#8782, 16#8783, 16#8785, 16#8788, 16#878B, 16#878D, 16#8793, 16#8797, 16#879F, 16#87A8, 16#87AB, 16#87AC, 16#87AD, 16#87AF, 16#87B3, 16#87B5, 16#87BA, 16#87BD, 16#87C0, 16#87C6, 16#87CA, 16#87CB, 16#87D1, 16#87D2, 16#87D3, 16#87DB, 16#87E0, 16#87E5, 16#87EA, 16#87EE, 16#87F9, 16#87FE, 16#8803, 16#880A, 16#8813, 16#8815, 16#8816, 16#881B, 16#8821, 16#8822, 16#8832, 16#8839, 16#883C, 16#8840, 16#8844, 16#8845, 16#884C, 16#884D, 16#8854, 16#8857, 16#8859, 16#8861, 16#8862, 16#8863, 16#8864, 16#8865, 16#8868, 16#8869, 16#886B, 16#886C, 16#886E, 16#8870, 16#8872, 16#8877, 16#887D, 16#887E, 16#887F, 16#8881, 16#8882, 16#8884, 16#8885, 16#8888, 16#888B, 16#888D, 16#8892, 16#8896, 16#889C, 16#88A2, 16#88A4, 16#88AB, 16#88AD, 16#88B1, 16#88B7, 16#88BC, 16#88C1, 16#88C2, 16#88C5, 16#88C6, 16#88C9, 16#88CE, 16#88D2, 16#88D4, 16#88D5, 16#88D8, 16#88D9, 16#88DF, 16#88E2, 16#88E3, 16#88E4, 16#88E5, 16#88E8, 16#88F0, 16#88F1, 16#88F3, 16#88F4, 16#88F8, 16#88F9, 16#88FC, 16#88FE, 16#8902, 16#890A, 16#8910, 16#8912, 16#8913, 16#8919, 16#891A, 16#891B, 16#8921, 16#8925, 16#892A, 16#892B, 16#8930, 16#8934, 16#8936, 16#8941, 16#8944, 16#895E, 16#895F, 16#8966, 16#897B, 16#897F, 16#8981, 16#8983, 16#8986, 16#89C1, 16#89C2, 16#89C4, 16#89C5, 16#89C6, 16#89C7, 16#89C8, 16#89C9, 16#89CA, 16#89CB, 16#89CC, 16#89CE, 16#89CF, 16#89D0, 16#89D1, 16#89D2, 16#89D6, 16#89DA, 16#89DC, 16#89DE, 16#89E3, 16#89E5, 16#89E6, 16#89EB, 16#89EF, 16#89F3, 16#8A00, 16#8A07, 16#8A3E, 16#8A48, 16#8A79, 16#8A89, 16#8A8A, 16#8A93, 16#8B07, 16#8B26, 16#8B66, 16#8B6C, 16#8BA0, 16#8BA1, 16#8BA2, 16#8BA3, 16#8BA4, 16#8BA5, 16#8BA6, 16#8BA7, 16#8BA8, 16#8BA9, 16#8BAA, 16#8BAB, 16#8BAD, 16#8BAE, 16#8BAF, 16#8BB0, 16#8BB2, 16#8BB3, 16#8BB4, 16#8BB5, 16#8BB6, 16#8BB7, 16#8BB8, 16#8BB9, 16#8BBA, 16#8BBC, 16#8BBD, 16#8BBE, 16#8BBF, 16#8BC0, 16#8BC1, 16#8BC2, 16#8BC3, 16#8BC4, 16#8BC5, 16#8BC6, 16#8BC8, 16#8BC9, 16#8BCA, 16#8BCB, 16#8BCC, 16#8BCD, 16#8BCE, 16#8BCF, 16#8BD1, 16#8BD2, 16#8BD3, 16#8BD4, 16#8BD5, 16#8BD6, 16#8BD7, 16#8BD8, 16#8BD9, 16#8BDA, 16#8BDB, 16#8BDC, 16#8BDD, 16#8BDE, 16#8BDF, 16#8BE0, 16#8BE1, 16#8BE2, 16#8BE3, 16#8BE4, 16#8BE5, 16#8BE6, 16#8BE7, 16#8BE8, 16#8BE9, 16#8BEB, 16#8BEC, 16#8BED, 16#8BEE, 16#8BEF, 16#8BF0, 16#8BF1, 16#8BF2, 16#8BF3, 16#8BF4, 16#8BF5, 16#8BF6, 16#8BF7, 16#8BF8, 16#8BF9, 16#8BFA, 16#8BFB, 16#8BFC, 16#8BFD, 16#8BFE, 16#8BFF, 16#8C00, 16#8C01, 16#8C02, 16#8C03, 16#8C04, 16#8C05, 16#8C06, 16#8C07, 16#8C08, 16#8C0A, 16#8C0B, 16#8C0C, 16#8C0D, 16#8C0E, 16#8C0F, 16#8C10, 16#8C11, 16#8C12, 16#8C13, 16#8C14, 16#8C15, 16#8C16, 16#8C17, 16#8C18, 16#8C19, 16#8C1A, 16#8C1B, 16#8C1C, 16#8C1D, 16#8C1F, 16#8C20, 16#8C21, 16#8C22, 16#8C23, 16#8C24, 16#8C25, 16#8C26, 16#8C27, 16#8C28, 16#8C29, 16#8C2A, 16#8C2B, 16#8C2C, 16#8C2D, 16#8C2E, 16#8C2F, 16#8C30, 16#8C31, 16#8C32, 16#8C33, 16#8C34, 16#8C35, 16#8C36, 16#8C37, 16#8C41, 16#8C46, 16#8C47, 16#8C49, 16#8C4C, 16#8C55, 16#8C5A, 16#8C61, 16#8C62, 16#8C6A, 16#8C6B, 16#8C73, 16#8C78, 16#8C79, 16#8C7A, 16#8C82, 16#8C85, 16#8C89, 16#8C8A, 16#8C8C, 16#8C94, 16#8C98, 16#8D1D, 16#8D1E, 16#8D1F, 16#8D21, 16#8D22, 16#8D23, 16#8D24, 16#8D25, 16#8D26, 16#8D27, 16#8D28, 16#8D29, 16#8D2A, 16#8D2B, 16#8D2C, 16#8D2D, 16#8D2E, 16#8D2F, 16#8D30, 16#8D31, 16#8D32, 16#8D33, 16#8D34, 16#8D35, 16#8D36, 16#8D37, 16#8D38, 16#8D39, 16#8D3A, 16#8D3B, 16#8D3C, 16#8D3D, 16#8D3E, 16#8D3F, 16#8D40, 16#8D41, 16#8D42, 16#8D43, 16#8D44, 16#8D45, 16#8D46, 16#8D47, 16#8D48, 16#8D49, 16#8D4A, 16#8D4B, 16#8D4C, 16#8D4D, 16#8D4E, 16#8D4F, 16#8D50, 16#8D53, 16#8D54, 16#8D55, 16#8D56, 16#8D58, 16#8D59, 16#8D5A, 16#8D5B, 16#8D5C, 16#8D5D, 16#8D5E, 16#8D60, 16#8D61, 16#8D62, 16#8D63, 16#8D64, 16#8D66, 16#8D67, 16#8D6B, 16#8D6D, 16#8D70, 16#8D73, 16#8D74, 16#8D75, 16#8D76, 16#8D77, 16#8D81, 16#8D84, 16#8D85, 16#8D8A, 16#8D8B, 16#8D91, 16#8D94, 16#8D9F, 16#8DA3, 16#8DB1, 16#8DB3, 16#8DB4, 16#8DB5, 16#8DB8, 16#8DBA, 16#8DBC, 16#8DBE, 16#8DBF, 16#8DC3, 16#8DC4, 16#8DC6, 16#8DCB, 16#8DCC, 16#8DCE, 16#8DCF, 16#8DD1, 16#8DD6, 16#8DD7, 16#8DDA, 16#8DDB, 16#8DDD, 16#8DDE, 16#8DDF, 16#8DE3, 16#8DE4, 16#8DE8, 16#8DEA, 16#8DEB, 16#8DEC, 16#8DEF, 16#8DF3, 16#8DF5, 16#8DF7, 16#8DF8, 16#8DF9, 16#8DFA, 16#8DFB, 16#8DFD, 16#8E05, 16#8E09, 16#8E0A, 16#8E0C, 16#8E0F, 16#8E14, 16#8E1D, 16#8E1E, 16#8E1F, 16#8E22, 16#8E23, 16#8E29, 16#8E2A, 16#8E2C, 16#8E2E, 16#8E2F, 16#8E31, 16#8E35, 16#8E39, 16#8E3A, 16#8E3D, 16#8E40, 16#8E41, 16#8E42, 16#8E44, 16#8E47, 16#8E48, 16#8E49, 16#8E4A, 16#8E4B, 16#8E51, 16#8E52, 16#8E59, 16#8E66, 16#8E69, 16#8E6C, 16#8E6D, 16#8E6F, 16#8E70, 16#8E72, 16#8E74, 16#8E76, 16#8E7C, 16#8E7F, 16#8E81, 16#8E85, 16#8E87, 16#8E8F, 16#8E90, 16#8E94, 16#8E9C, 16#8E9E, 16#8EAB, 16#8EAC, 16#8EAF, 16#8EB2, 16#8EBA, 16#8ECE, 16#8F66, 16#8F67, 16#8F68, 16#8F69, 16#8F6B, 16#8F6C, 16#8F6D, 16#8F6E, 16#8F6F, 16#8F70, 16#8F71, 16#8F72, 16#8F73, 16#8F74, 16#8F75, 16#8F76, 16#8F77, 16#8F78, 16#8F79, 16#8F7A, 16#8F7B, 16#8F7C, 16#8F7D, 16#8F7E, 16#8F7F, 16#8F81, 16#8F82, 16#8F83, 16#8F84, 16#8F85, 16#8F86, 16#8F87, 16#8F88, 16#8F89, 16#8F8A, 16#8F8B, 16#8F8D, 16#8F8E, 16#8F8F, 16#8F90, 16#8F91, 16#8F93, 16#8F94, 16#8F95, 16#8F96, 16#8F97, 16#8F98, 16#8F99, 16#8F9A, 16#8F9B, 16#8F9C, 16#8F9E, 16#8F9F, 16#8FA3, 16#8FA8, 16#8FA9, 16#8FAB, 16#8FB0, 16#8FB1, 16#8FB6, 16#8FB9, 16#8FBD, 16#8FBE, 16#8FC1, 16#8FC2, 16#8FC4, 16#8FC5, 16#8FC7, 16#8FC8, 16#8FCE, 16#8FD0, 16#8FD1, 16#8FD3, 16#8FD4, 16#8FD5, 16#8FD8, 16#8FD9, 16#8FDB, 16#8FDC, 16#8FDD, 16#8FDE, 16#8FDF, 16#8FE2, 16#8FE4, 16#8FE5, 16#8FE6, 16#8FE8, 16#8FE9, 16#8FEA, 16#8FEB, 16#8FED, 16#8FEE, 16#8FF0, 16#8FF3, 16#8FF7, 16#8FF8, 16#8FF9, 16#8FFD, 16#9000, 16#9001, 16#9002, 16#9003, 16#9004, 16#9005, 16#9006, 16#9009, 16#900A, 16#900B, 16#900D, 16#900F, 16#9010, 16#9011, 16#9012, 16#9014, 16#9016, 16#9017, 16#901A, 16#901B, 16#901D, 16#901E, 16#901F, 16#9020, 16#9021, 16#9022, 16#9026, 16#902D, 16#902E, 16#902F, 16#9035, 16#9036, 16#9038, 16#903B, 16#903C, 16#903E, 16#9041, 16#9042, 16#9044, 16#9047, 16#904D, 16#904F, 16#9050, 16#9051, 16#9052, 16#9053, 16#9057, 16#9058, 16#905B, 16#9062, 16#9063, 16#9065, 16#9068, 16#906D, 16#906E, 16#9074, 16#9075, 16#907D, 16#907F, 16#9080, 16#9082, 16#9083, 16#9088, 16#908B, 16#9091, 16#9093, 16#9095, 16#9097, 16#9099, 16#909B, 16#909D, 16#90A1, 16#90A2, 16#90A3, 16#90A6, 16#90AA, 16#90AC, 16#90AE, 16#90AF, 16#90B0, 16#90B1, 16#90B3, 16#90B4, 16#90B5, 16#90B6, 16#90B8, 16#90B9, 16#90BA, 16#90BB, 16#90BE, 16#90C1, 16#90C4, 16#90C5, 16#90C7, 16#90CA, 16#90CE, 16#90CF, 16#90D0, 16#90D1, 16#90D3, 16#90D7, 16#90DB, 16#90DC, 16#90DD, 16#90E1, 16#90E2, 16#90E6, 16#90E7, 16#90E8, 16#90EB, 16#90ED, 16#90EF, 16#90F4, 16#90F8, 16#90FD, 16#90FE, 16#9102, 16#9104, 16#9119, 16#911E, 16#9122, 16#9123, 16#912F, 16#9131, 16#9139, 16#9143, 16#9146, 16#9149, 16#914A, 16#914B, 16#914C, 16#914D, 16#914E, 16#914F, 16#9150, 16#9152, 16#9157, 16#915A, 16#915D, 16#915E, 16#9161, 16#9162, 16#9163, 16#9164, 16#9165, 16#9169, 16#916A, 16#916C, 16#916E, 16#916F, 16#9170, 16#9171, 16#9172, 16#9174, 16#9175, 16#9176, 16#9177, 16#9178, 16#9179, 16#917D, 16#917E, 16#917F, 16#9185, 16#9187, 16#9189, 16#918B, 16#918C, 16#918D, 16#9190, 16#9191, 16#9192, 16#919A, 16#919B, 16#91A2, 16#91A3, 16#91AA, 16#91AD, 16#91AE, 16#91AF, 16#91B4, 16#91B5, 16#91BA, 16#91C7, 16#91C9, 16#91CA, 16#91CC, 16#91CD, 16#91CE, 16#91CF, 16#91D1, 16#91DC, 16#9274, 16#928E, 16#92AE, 16#92C8, 16#933E, 16#936A, 16#938F, 16#93CA, 16#93D6, 16#943E, 16#946B, 16#9485, 16#9486, 16#9487, 16#9488, 16#9489, 16#948A, 16#948B, 16#948C, 16#948D, 16#948E, 16#948F, 16#9490, 16#9492, 16#9493, 16#9494, 16#9495, 16#9497, 16#9499, 16#949A, 16#949B, 16#949C, 16#949D, 16#949E, 16#949F, 16#94A0, 16#94A1, 16#94A2, 16#94A3, 16#94A4, 16#94A5, 16#94A6, 16#94A7, 16#94A8, 16#94A9, 16#94AA, 16#94AB, 16#94AC, 16#94AD, 16#94AE, 16#94AF, 16#94B0, 16#94B1, 16#94B2, 16#94B3, 16#94B4, 16#94B5, 16#94B6, 16#94B7, 16#94B8, 16#94B9, 16#94BA, 16#94BB, 16#94BC, 16#94BD, 16#94BE, 16#94BF, 16#94C0, 16#94C1, 16#94C2, 16#94C3, 16#94C4, 16#94C5, 16#94C6, 16#94C8, 16#94C9, 16#94CA, 16#94CB, 16#94CC, 16#94CD, 16#94CE, 16#94D0, 16#94D1, 16#94D2, 16#94D5, 16#94D6, 16#94D7, 16#94D8, 16#94D9, 16#94DB, 16#94DC, 16#94DD, 16#94DE, 16#94DF, 16#94E0, 16#94E1, 16#94E2, 16#94E3, 16#94E4, 16#94E5, 16#94E7, 16#94E8, 16#94E9, 16#94EA, 16#94EB, 16#94EC, 16#94ED, 16#94EE, 16#94EF, 16#94F0, 16#94F1, 16#94F2, 16#94F3, 16#94F4, 16#94F5, 16#94F6, 16#94F7, 16#94F8, 16#94F9, 16#94FA, 16#94FC, 16#94FD, 16#94FE, 16#94FF, 16#9500, 16#9501, 16#9502, 16#9503, 16#9504, 16#9505, 16#9506, 16#9507, 16#9508, 16#9509, 16#950A, 16#950B, 16#950C, 16#950D, 16#950E, 16#950F, 16#9510, 16#9511, 16#9512, 16#9513, 16#9514, 16#9515, 16#9516, 16#9517, 16#9518, 16#9519, 16#951A, 16#951B, 16#951D, 16#951E, 16#951F, 16#9521, 16#9522, 16#9523, 16#9524, 16#9525, 16#9526, 16#9528, 16#9529, 16#952A, 16#952B, 16#952C, 16#952D, 16#952E, 16#952F, 16#9530, 16#9531, 16#9532, 16#9534, 16#9535, 16#9536, 16#9537, 16#9538, 16#9539, 16#953A, 16#953B, 16#953C, 16#953E, 16#953F, 16#9540, 16#9541, 16#9542, 16#9544, 16#9545, 16#9546, 16#9547, 16#9549, 16#954A, 16#954C, 16#954D, 16#954E, 16#954F, 16#9550, 16#9551, 16#9552, 16#9553, 16#9554, 16#9556, 16#9557, 16#9558, 16#9559, 16#955B, 16#955C, 16#955D, 16#955E, 16#955F, 16#9561, 16#9562, 16#9563, 16#9564, 16#9565, 16#9566, 16#9567, 16#9568, 16#9569, 16#956A, 16#956B, 16#956C, 16#956D, 16#956F, 16#9570, 16#9571, 16#9572, 16#9573, 16#9576, 16#957F, 16#95E8, 16#95E9, 16#95EA, 16#95EB, 16#95ED, 16#95EE, 16#95EF, 16#95F0, 16#95F1, 16#95F2, 16#95F3, 16#95F4, 16#95F5, 16#95F6, 16#95F7, 16#95F8, 16#95F9, 16#95FA, 16#95FB, 16#95FC, 16#95FD, 16#95FE, 16#9600, 16#9601, 16#9602, 16#9603, 16#9604, 16#9605, 16#9606, 16#9608, 16#9609, 16#960A, 16#960B, 16#960C, 16#960D, 16#960E, 16#960F, 16#9610, 16#9611, 16#9612, 16#9614, 16#9615, 16#9616, 16#9617, 16#9619, 16#961A, 16#961C, 16#961D, 16#961F, 16#9621, 16#9622, 16#962A, 16#962E, 16#9631, 16#9632, 16#9633, 16#9634, 16#9635, 16#9636, 16#963B, 16#963C, 16#963D, 16#963F, 16#9640, 16#9642, 16#9644, 16#9645, 16#9646, 16#9647, 16#9648, 16#9649, 16#964B, 16#964C, 16#964D, 16#9650, 16#9654, 16#9655, 16#965B, 16#965F, 16#9661, 16#9662, 16#9664, 16#9667, 16#9668, 16#9669, 16#966A, 16#966C, 16#9672, 16#9674, 16#9675, 16#9676, 16#9677, 16#9685, 16#9686, 16#9688, 16#968B, 16#968D, 16#968F, 16#9690, 16#9694, 16#9697, 16#9698, 16#9699, 16#969C, 16#96A7, 16#96B0, 16#96B3, 16#96B6, 16#96B9, 16#96BC, 16#96BD, 16#96BE, 16#96C0, 16#96C1, 16#96C4, 16#96C5, 16#96C6, 16#96C7, 16#96C9, 16#96CC, 16#96CD, 16#96CE, 16#96CF, 16#96D2, 16#96D5, 16#96E0, 16#96E8, 16#96E9, 16#96EA, 16#96EF, 16#96F3, 16#96F6, 16#96F7, 16#96F9, 16#96FE, 16#9700, 16#9701, 16#9704, 16#9706, 16#9707, 16#9708, 16#9709, 16#970D, 16#970E, 16#970F, 16#9713, 16#9716, 16#971C, 16#971E, 16#972A, 16#972D, 16#9730, 16#9732, 16#9738, 16#9739, 16#973E, 16#9752, 16#9753, 16#9756, 16#9759, 16#975B, 16#975E, 16#9760, 16#9761, 16#9762, 16#9765, 16#9769, 16#9773, 16#9774, 16#9776, 16#977C, 16#9785, 16#978B, 16#978D, 16#9791, 16#9792, 16#9794, 16#9798, 16#97A0, 16#97A3, 16#97AB, 16#97AD, 16#97AF, 16#97B2, 16#97B4, 16#97E6, 16#97E7, 16#97E9, 16#97EA, 16#97EB, 16#97EC, 16#97ED, 16#97F3, 16#97F5, 16#97F6, 16#9875, 16#9876, 16#9877, 16#9878, 16#9879, 16#987A, 16#987B, 16#987C, 16#987D, 16#987E, 16#987F, 16#9880, 16#9881, 16#9882, 16#9883, 16#9884, 16#9885, 16#9886, 16#9887, 16#9888, 16#9889, 16#988A, 16#988C, 16#988D, 16#988F, 16#9890, 16#9891, 16#9893, 16#9894, 16#9896, 16#9897, 16#9898, 16#989A, 16#989B, 16#989C, 16#989D, 16#989E, 16#989F, 16#98A0, 16#98A1, 16#98A2, 16#98A4, 16#98A5, 16#98A6, 16#98A7, 16#98CE, 16#98D1, 16#98D2, 16#98D3, 16#98D5, 16#98D8, 16#98D9, 16#98DA, 16#98DE, 16#98DF, 16#98E7, 16#98E8, 16#990D, 16#9910, 16#992E, 16#9954, 16#9955, 16#9963, 16#9965, 16#9967, 16#9968, 16#9969, 16#996A, 16#996B, 16#996C, 16#996D, 16#996E, 16#996F, 16#9970, 16#9971, 16#9972, 16#9974, 16#9975, 16#9976, 16#9977, 16#997A, 16#997C, 16#997D, 16#997F, 16#9980, 16#9981, 16#9984, 16#9985, 16#9986, 16#9987, 16#9988, 16#998A, 16#998B, 16#998D, 16#998F, 16#9990, 16#9991, 16#9992, 16#9993, 16#9994, 16#9995, 16#9996, 16#9997, 16#9998, 16#9999, 16#99A5, 16#99A8, 16#9A6C, 16#9A6D, 16#9A6E, 16#9A6F, 16#9A70, 16#9A71, 16#9A73, 16#9A74, 16#9A75, 16#9A76, 16#9A77, 16#9A78, 16#9A79, 16#9A7A, 16#9A7B, 16#9A7C, 16#9A7D, 16#9A7E, 16#9A7F, 16#9A80, 16#9A81, 16#9A82, 16#9A84, 16#9A85, 16#9A86, 16#9A87, 16#9A88, 16#9A8A, 16#9A8B, 16#9A8C, 16#9A8F, 16#9A90, 16#9A91, 16#9A92, 16#9A93, 16#9A96, 16#9A97, 16#9A98, 16#9A9A, 16#9A9B, 16#9A9C, 16#9A9D, 16#9A9E, 16#9A9F, 16#9AA0, 16#9AA1, 16#9AA2, 16#9AA3, 16#9AA4, 16#9AA5, 16#9AA7, 16#9AA8, 16#9AB0, 16#9AB1, 16#9AB6, 16#9AB7, 16#9AB8, 16#9ABA, 16#9ABC, 16#9AC0, 16#9AC1, 16#9AC2, 16#9AC5, 16#9ACB, 16#9ACC, 16#9AD1, 16#9AD3, 16#9AD8, 16#9ADF, 16#9AE1, 16#9AE6, 16#9AEB, 16#9AED, 16#9AEF, 16#9AF9, 16#9AFB, 16#9B03, 16#9B08, 16#9B0F, 16#9B13, 16#9B1F, 16#9B23, 16#9B2F, 16#9B32, 16#9B3B, 16#9B3C, 16#9B41, 16#9B42, 16#9B43, 16#9B44, 16#9B45, 16#9B47, 16#9B48, 16#9B49, 16#9B4D, 16#9B4F, 16#9B51, 16#9B54, 16#9C7C, 16#9C7F, 16#9C81, 16#9C82, 16#9C85, 16#9C86, 16#9C87, 16#9C88, 16#9C8B, 16#9C8D, 16#9C8E, 16#9C90, 16#9C91, 16#9C92, 16#9C94, 16#9C95, 16#9C9A, 16#9C9B, 16#9C9C, 16#9C9E, 16#9C9F, 16#9CA0, 16#9CA1, 16#9CA2, 16#9CA3, 16#9CA4, 16#9CA5, 16#9CA6, 16#9CA7, 16#9CA8, 16#9CA9, 16#9CAB, 16#9CAD, 16#9CAE, 16#9CB0, 16#9CB1, 16#9CB2, 16#9CB3, 16#9CB4, 16#9CB5, 16#9CB6, 16#9CB7, 16#9CB8, 16#9CBA, 16#9CBB, 16#9CBC, 16#9CBD, 16#9CC3, 16#9CC4, 16#9CC5, 16#9CC6, 16#9CC7, 16#9CCA, 16#9CCB, 16#9CCC, 16#9CCD, 16#9CCE, 16#9CCF, 16#9CD0, 16#9CD3, 16#9CD4, 16#9CD5, 16#9CD6, 16#9CD7, 16#9CD8, 16#9CD9, 16#9CDC, 16#9CDD, 16#9CDE, 16#9CDF, 16#9CE2, 16#9E1F, 16#9E20, 16#9E21, 16#9E22, 16#9E23, 16#9E25, 16#9E26, 16#9E28, 16#9E29, 16#9E2A, 16#9E2B, 16#9E2C, 16#9E2D, 16#9E2F, 16#9E31, 16#9E32, 16#9E33, 16#9E35, 16#9E36, 16#9E37, 16#9E38, 16#9E39, 16#9E3A, 16#9E3D, 16#9E3E, 16#9E3F, 16#9E41, 16#9E42, 16#9E43, 16#9E44, 16#9E45, 16#9E46, 16#9E47, 16#9E48, 16#9E49, 16#9E4A, 16#9E4B, 16#9E4C, 16#9E4E, 16#9E4F, 16#9E51, 16#9E55, 16#9E57, 16#9E58, 16#9E5A, 16#9E5B, 16#9E5C, 16#9E5E, 16#9E63, 16#9E64, 16#9E66, 16#9E67, 16#9E68, 16#9E69, 16#9E6A, 16#9E6B, 16#9E6C, 16#9E6D, 16#9E70, 16#9E71, 16#9E73, 16#9E7E, 16#9E7F, 16#9E82, 16#9E87, 16#9E88, 16#9E8B, 16#9E92, 16#9E93, 16#9E9D, 16#9E9F, 16#9EA6, 16#9EB4, 16#9EB8, 16#9EBB, 16#9EBD, 16#9EBE, 16#9EC4, 16#9EC9, 16#9ECD, 16#9ECE, 16#9ECF, 16#9ED1, 16#9ED4, 16#9ED8, 16#9EDB, 16#9EDC, 16#9EDD, 16#9EDF, 16#9EE0, 16#9EE2, 16#9EE5, 16#9EE7, 16#9EE9, 16#9EEA, 16#9EEF, 16#9EF9, 16#9EFB, 16#9EFC, 16#9EFE, 16#9F0B, 16#9F0D, 16#9F0E, 16#9F10, 16#9F13, 16#9F17, 16#9F19, 16#9F20, 16#9F22, 16#9F2C, 16#9F2F, 16#9F37, 16#9F39, 16#9F3B, 16#9F3D, 16#9F3E, 16#9F44, 16#9F50, 16#9F51, 16#9F7F, 16#9F80, 16#9F83, 16#9F84, 16#9F85, 16#9F86, 16#9F87, 16#9F88, 16#9F89, 16#9F8A, 16#9F8B, 16#9F8C, 16#9F99, 16#9F9A, 16#9F9B, 16#9F9F, 16#9FA0, 16#FE31, 16#FE33, 16#FE34, 16#FE35, 16#FE36, 16#FE37, 16#FE38, 16#FE39, 16#FE3A, 16#FE3B, 16#FE3C, 16#FE3D, 16#FE3E, 16#FE3F, 16#FE40, 16#FE41, 16#FE42, 16#FE43, 16#FE44, 16#FF01, 16#FF02, 16#FF03, 16#FF04, 16#FF05, 16#FF06, 16#FF07, 16#FF08, 16#FF09, 16#FF0A, 16#FF0B, 16#FF0C, 16#FF0D, 16#FF0E, 16#FF0F, 16#FF10, 16#FF11, 16#FF12, 16#FF13, 16#FF14, 16#FF15, 16#FF16, 16#FF17, 16#FF18, 16#FF19, 16#FF1A, 16#FF1B, 16#FF1C, 16#FF1D, 16#FF1E, 16#FF1F, 16#FF20, 16#FF21, 16#FF22, 16#FF23, 16#FF24, 16#FF25, 16#FF26, 16#FF27, 16#FF28, 16#FF29, 16#FF2A, 16#FF2B, 16#FF2C, 16#FF2D, 16#FF2E, 16#FF2F, 16#FF30, 16#FF31, 16#FF32, 16#FF33, 16#FF34, 16#FF35, 16#FF36, 16#FF37, 16#FF38, 16#FF39, 16#FF3A, 16#FF3B, 16#FF3C, 16#FF3D, 16#FF3E, 16#FF3F, 16#FF40, 16#FF41, 16#FF42, 16#FF43, 16#FF44, 16#FF45, 16#FF46, 16#FF47, 16#FF48, 16#FF49, 16#FF4A, 16#FF4B, 16#FF4C, 16#FF4D, 16#FF4E, 16#FF4F, 16#FF50, 16#FF51, 16#FF52, 16#FF53, 16#FF54, 16#FF55, 16#FF56, 16#FF57, 16#FF58, 16#FF59, 16#FF5A, 16#FF5B, 16#FF5C, 16#FF5D, 16#FF5E, 16#FFE0, 16#FFE1, 16#FFE3, 16#FFE5, 2(0)];
